// TIA Portal V20 export
// export: Created 2025-12-01T14:56:51.5395909Z, ExportSetting None, DisplayName Totally Integrated Automation Portal, DisplayVersion V20 Update 3, DisplayName TIA Portal Openness, DisplayVersion V20 Update 3, DisplayName TIA Portal Version Control Interface, DisplayVersion V20 Update 3, DisplayName STEP 7 Professional, DisplayVersion V20 Update 3, DisplayName STEP 7 Safety, DisplayVersion V20 Update 2, DisplayName WinCC Basic/Comfort/Advanced, DisplayVersion V20 Update 3, DisplayName WinCC Professional, DisplayVersion V20 Update 3, DisplayName WinCC Unified, DisplayVersion V20 Update 3
FUNCTION_BLOCK "FB351_DesRemontador_Remontador_Horquilla"   // FB351, LAD
TITLE = Control del Ramal de Salidas
{ S7_Optimized_Access := 'FALSE' }
AUTHOR : REFORMAR
NAME : 20160211
VERSION : 3.1
// Dani Palacios: Modificación octubre 2017 para poder desabilitar la maquina con un bit (por ejemplo en la puesta a punto si no esta montada o en el simulador)
// La modificación esta sin probar y es todo lo relativo a la variable Maquina_Desabilitada
// (bloqueo evolución desde etapa 0, bloqueo activación salidas en etapa 0 , fin vi sin mirar detectores y activación posición de reposo sin mirar detectores y variabkles de fin de movimiento).
// ES RESPONSABILIDAD DEL QUE DESABILITA LA MAQUINA QUE ESTA ESTE EN UNA POSICION QUE PERMITA EL MOVIMIENTO DE LAS CARGAS A TRAVES DE ELLA
// stored: AutoNumber false, SetENOAutomatically false
   VAR_INPUT
      Maquina : UInt;   // Numero de Maquina (Mesa)
      Error_Tx : Bool;   // Error en el Tx
      EnTension : Bool;   // Existe Tension en la Mesa
      MAQx_Desabilitada : Bool;   // Config MAQ. >>> DesHabilitada
      TipoPaleta : Bool;   // Si 1, EUR. Si 0, medio paleta
      Termico_Elevacion : Bool;   // Termico de la Elevacion
      Termico_Horquilla : Bool;   // Termico de la Horquilla
      ParElevacion_ErrorRotura : Bool;
      pHsMx : Bool;   // pHs de la Mesa
      EnMovimiento_Tx : Bool;   // En Movimiento Tx
      ELEV_SegUp : Bool;   // ELEV >> Seguridad Up
      ELEV_SegDw : Bool;   // ELEV >> Seguridad Down
      ELEV_PosUp : Bool;   // ELEV >> Posicion Up
      ELEV_PosMid : Bool;   // ELEV >> Posicion Midle
      ELEV_PosDw : Bool;   // ELEV >> Posicion Down
      ELEV_EnMovimiento : Bool;   // ELEV >> En Movimiento
      HORQ_SegRecogida : Bool;   // HORQ >> Seguridad Atras
      HORQ_SegExtendida : Bool;   // HORQ >> Seguridad Adelante
      HORQ_Recogida : Bool;   // HORQ >> Posicion Atras
      HORQ_Medio : Bool;   // HORQ >> Posicion Medio
      HORQ_Extendida : Bool;   // HORQ >> Posicion Adelante
      HORQ_CV_Recogida : Bool;   // HORQ >> Cambio de Velocidad Atras
      HORQ_CV_Medio : Bool;   // HORQ >> Cambio de Velocidad Medio
      HORQ_CV_Extendida : Bool;   // HORQ >> Cambio de Velocidad Adelante
      HORQ_EnMovimiento : Bool;   // HORQ >> En Movimiento
      Elev_Carga_OK : Bool;
      RH_PasarReposo : Bool;   // Interlock >> Pasar a Reposo
      RH_SubirPaleta : Bool;   // Interlock >> Subir Paleta
      RH_DejarPaleta : Bool;   // Interlock >> Dejar Paleta
      RH_RemontarPaleta : Bool;   // Interlock >> Remontar Paleta
      RH_DesRemontarPaleta : Bool;   // Interlock >> DesRemontar Paleta
      V_TIM_EstabilidadMov : Time;   // TIM de Estabilidad de los Mov.
      V_TOut_Elevacion : Int := 7000;   // TimeOut del Mov. de Elevacion
      V_TOut_Horquillado : Int := 7000;   // TimeOut del Mov. de Horquillado
   END_VAR
   VAR_OUTPUT
      RH_Quieto : Bool;   // Interlock >> Quieto
      RH_FinMovimiento : Bool;   // Interlock >> Fin del Movimiento
   END_VAR
   VAR
      Rh_ET00 : Bool;
      Rh_ET100 : Bool;
      Rh_ET101 : Bool;
      Rh_ET102 : Bool;
      Rh_ET103 : Bool;
      Rh_ET104 : Bool;
      Rh_ET105 : Bool;
      Rh_ET106 : Bool;
      Rh_ET107 : Bool;
      Rh_ET108 : Bool;
      Rh_ET109 : Bool;
      Rh_ET11 : Bool;
      Rh_ET12 : Bool;
      Rh_ET13 : Bool;
      Rh_ET14 : Bool;
      Rh_ET15 : Bool;
      Rh_ET16 : Bool;
      Rh_ET21 : Bool;
      Rh_ET22 : Bool;
      Rh_ET23 : Bool;
      Rh_ET24 : Bool;
      Rh_ET31 : Bool;
      Rh_ET32 : Bool;
      Rh_ET41 : Bool;
      Rh_ET42 : Bool;
      Rh_ET43 : Bool;
      Rh_ET44 : Bool;
      Rh_ET51 : Bool;
      Rh_ET52 : Bool;
      Rh_ET53 : Bool;
      PosicionConocida : Bool;
      STAT_Quieto : Bool;   // Interna >> Quieto la Maquina
      STAT_FinMovimiento : Bool;   // Interna >> Fin de Movimiento
      CambioDir_SubidaBajada : Bool;   // Interna >> Cambio de Dir. Subida o Bajada
      MA_Ir_Up : Bool;
      MA_Ir_Dw : Bool;
      MA_Ir_Mid_Bajando : Bool;
      MA_Ir_Mid_Subiendo : Bool;
      MA_Ir_Adelante : Bool;
      MA_Ir_Atras : Bool;
      HORQ_VelocidadRapida : Bool;
      TIM_EstabilidadMov { S7_SetPoint := 'True'} : TON_TIME;
      TMP_EnTension { S7_SetPoint := 'True'} : "FB910_CNT_UHS";
      TOut_Elevacion { S7_SetPoint := 'True'} : "FB910_CNT_UHS";
      TOut_Horquillado { S7_SetPoint := 'True'} : "FB910_CNT_UHS";
      Manual : "MoviManualMaquina_Remontador";
   END_VAR
   VAR_TEMP
      EstadoZona : "EstadoZona";   // Estado de Zona de la Mesa
      EstadoMAQ : "EstadoMaquina_Remontador";   // Estado del Vehiculo Inteliguente de la Maquina
      Aux_ET00 : Bool;
   END_VAR
BEGIN

REGION Network 1: INICIALIZAR - Recoger las Variables de Estado de la Maquina
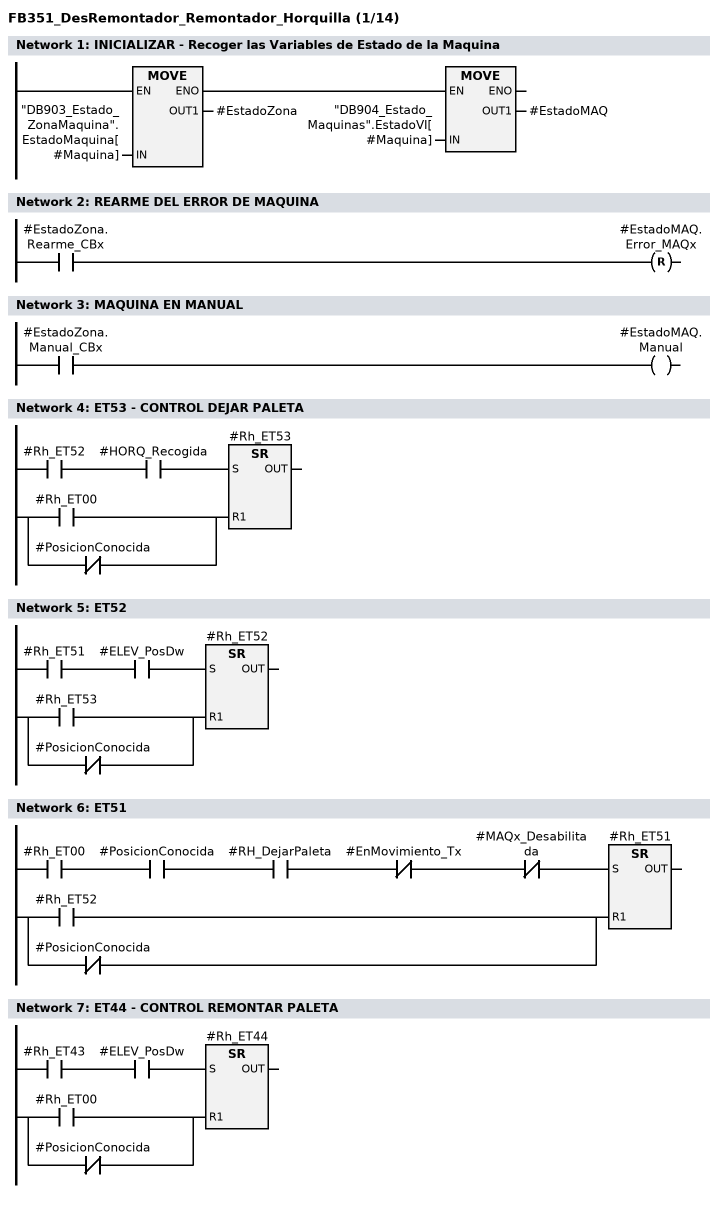
   RUNG wire#powerrail
      Move(in := "DB903_Estado_ZonaMaquina".EstadoMaquina[#Maquina], out1 => #EstadoZona)
      Move(in := "DB904_Estado_Maquinas".EstadoVI[#Maquina], out1 => #EstadoMAQ)
   END_RUNG
   // the same network as SCL:
   #EstadoZona := "DB903_Estado_ZonaMaquina".EstadoMaquina[#Maquina];
   #EstadoMAQ := "DB904_Estado_Maquinas".EstadoVI[#Maquina];
END_REGION

REGION Network 2: REARME DEL ERROR DE MAQUINA
   RUNG wire#powerrail
      Contact( #EstadoZona.Rearme_CBx )
      R_Coil( #EstadoMAQ.Error_MAQx )
   END_RUNG
   // the same network as SCL:
   IF #EstadoZona.Rearme_CBx THEN #EstadoMAQ.Error_MAQx := FALSE; END_IF;
END_REGION

REGION Network 3: MAQUINA EN MANUAL
   RUNG wire#powerrail
      Contact( #EstadoZona.Manual_CBx )
      Coil( #EstadoMAQ.Manual )
   END_RUNG
   // the same network as SCL:
   #EstadoMAQ.Manual := #EstadoZona.Manual_CBx;
END_REGION

REGION Network 4: ET53 - CONTROL DEJAR PALETA
   RUNG wire#powerrail
      Contact( #Rh_ET52 )
      Contact( #HORQ_Recogida )
      S_SR(operand := #Rh_ET53, r1 := wire#w1)
   END_RUNG
   RUNG wire#powerrail
      Contact( #Rh_ET00 )
   END_RUNG wire#w1
   RUNG wire#powerrail
      I_Contact( #PosicionConocida )
   END_RUNG wire#w1
   // the same network as SCL:
   IF #Rh_ET52 AND #HORQ_Recogida THEN
       #Rh_ET53 := TRUE;   // SR flip-flop
   END_IF;
   IF #Rh_ET00 OR NOT #PosicionConocida THEN #Rh_ET53 := FALSE; END_IF;
END_REGION

REGION Network 5: ET52
   RUNG wire#powerrail
      Contact( #Rh_ET51 )
      Contact( #ELEV_PosDw )
      S_SR(operand := #Rh_ET52, r1 := wire#w1)
   END_RUNG
   RUNG wire#powerrail
      Contact( #Rh_ET53 )
   END_RUNG wire#w1
   RUNG wire#powerrail
      I_Contact( #PosicionConocida )
   END_RUNG wire#w1
   // the same network as SCL:
   IF #Rh_ET51 AND #ELEV_PosDw THEN
       #Rh_ET52 := TRUE;   // SR flip-flop
   END_IF;
   IF #Rh_ET53 OR NOT #PosicionConocida THEN #Rh_ET52 := FALSE; END_IF;
END_REGION

REGION Network 6: ET51
   RUNG wire#powerrail
      Contact( #Rh_ET00 )
      Contact( #PosicionConocida )
      Contact( #RH_DejarPaleta )
      I_Contact( #EnMovimiento_Tx )
      I_Contact( #MAQx_Desabilitada )
      S_SR(operand := #Rh_ET51, r1 := wire#w1)
   END_RUNG
   RUNG wire#powerrail
      Contact( #Rh_ET52 )
   END_RUNG wire#w1
   RUNG wire#powerrail
      I_Contact( #PosicionConocida )
   END_RUNG wire#w1
   // the same network as SCL:
   IF #Rh_ET00 AND #PosicionConocida AND #RH_DejarPaleta AND NOT #EnMovimiento_Tx AND NOT #MAQx_Desabilitada THEN
       #Rh_ET51 := TRUE;   // SR flip-flop
   END_IF;
   IF #Rh_ET52 OR NOT #PosicionConocida THEN #Rh_ET51 := FALSE; END_IF;
END_REGION

REGION Network 7: ET44 - CONTROL REMONTAR PALETA
   RUNG wire#powerrail
      Contact( #Rh_ET43 )
      Contact( #ELEV_PosDw )
      S_SR(operand := #Rh_ET44, r1 := wire#w1)
   END_RUNG
   RUNG wire#powerrail
      Contact( #Rh_ET00 )
   END_RUNG wire#w1
   RUNG wire#powerrail
      I_Contact( #PosicionConocida )
   END_RUNG wire#w1
   // the same network as SCL:
   IF #Rh_ET43 AND #ELEV_PosDw THEN
       #Rh_ET44 := TRUE;   // SR flip-flop
   END_IF;
   IF #Rh_ET00 OR NOT #PosicionConocida THEN #Rh_ET44 := FALSE; END_IF;
END_REGION

REGION Network 8: ET43
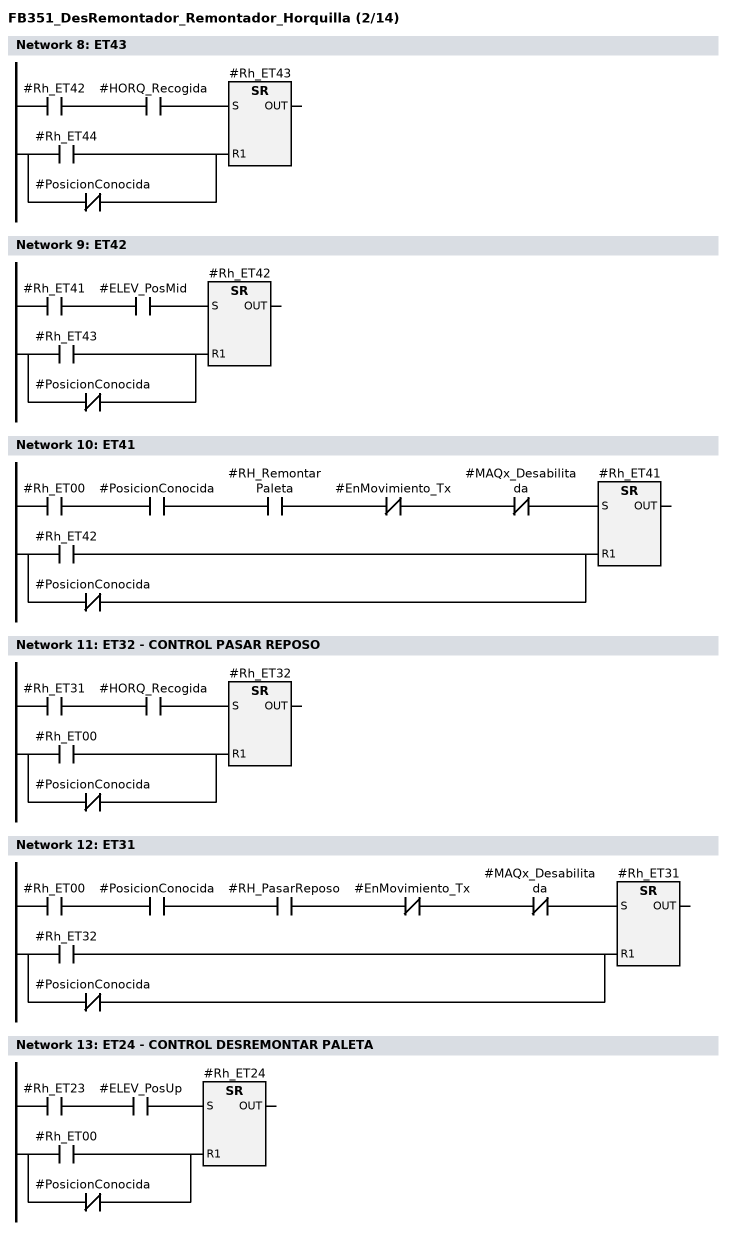
   RUNG wire#powerrail
      Contact( #Rh_ET42 )
      Contact( #HORQ_Recogida )
      S_SR(operand := #Rh_ET43, r1 := wire#w1)
   END_RUNG
   RUNG wire#powerrail
      Contact( #Rh_ET44 )
   END_RUNG wire#w1
   RUNG wire#powerrail
      I_Contact( #PosicionConocida )
   END_RUNG wire#w1
   // the same network as SCL:
   IF #Rh_ET42 AND #HORQ_Recogida THEN
       #Rh_ET43 := TRUE;   // SR flip-flop
   END_IF;
   IF #Rh_ET44 OR NOT #PosicionConocida THEN #Rh_ET43 := FALSE; END_IF;
END_REGION

REGION Network 9: ET42
   RUNG wire#powerrail
      Contact( #Rh_ET41 )
      Contact( #ELEV_PosMid )
      S_SR(operand := #Rh_ET42, r1 := wire#w1)
   END_RUNG
   RUNG wire#powerrail
      Contact( #Rh_ET43 )
   END_RUNG wire#w1
   RUNG wire#powerrail
      I_Contact( #PosicionConocida )
   END_RUNG wire#w1
   // the same network as SCL:
   IF #Rh_ET41 AND #ELEV_PosMid THEN
       #Rh_ET42 := TRUE;   // SR flip-flop
   END_IF;
   IF #Rh_ET43 OR NOT #PosicionConocida THEN #Rh_ET42 := FALSE; END_IF;
END_REGION

REGION Network 10: ET41
   RUNG wire#powerrail
      Contact( #Rh_ET00 )
      Contact( #PosicionConocida )
      Contact( #RH_RemontarPaleta )
      I_Contact( #EnMovimiento_Tx )
      I_Contact( #MAQx_Desabilitada )
      S_SR(operand := #Rh_ET41, r1 := wire#w1)
   END_RUNG
   RUNG wire#powerrail
      Contact( #Rh_ET42 )
   END_RUNG wire#w1
   RUNG wire#powerrail
      I_Contact( #PosicionConocida )
   END_RUNG wire#w1
   // the same network as SCL:
   IF #Rh_ET00 AND #PosicionConocida AND #RH_RemontarPaleta AND NOT #EnMovimiento_Tx AND NOT #MAQx_Desabilitada THEN
       #Rh_ET41 := TRUE;   // SR flip-flop
   END_IF;
   IF #Rh_ET42 OR NOT #PosicionConocida THEN #Rh_ET41 := FALSE; END_IF;
END_REGION

REGION Network 11: ET32 - CONTROL PASAR REPOSO
   RUNG wire#powerrail
      Contact( #Rh_ET31 )
      Contact( #HORQ_Recogida )
      S_SR(operand := #Rh_ET32, r1 := wire#w1)
   END_RUNG
   RUNG wire#powerrail
      Contact( #Rh_ET00 )
   END_RUNG wire#w1
   RUNG wire#powerrail
      I_Contact( #PosicionConocida )
   END_RUNG wire#w1
   // the same network as SCL:
   IF #Rh_ET31 AND #HORQ_Recogida THEN
       #Rh_ET32 := TRUE;   // SR flip-flop
   END_IF;
   IF #Rh_ET00 OR NOT #PosicionConocida THEN #Rh_ET32 := FALSE; END_IF;
END_REGION

REGION Network 12: ET31
   RUNG wire#powerrail
      Contact( #Rh_ET00 )
      Contact( #PosicionConocida )
      Contact( #RH_PasarReposo )
      I_Contact( #EnMovimiento_Tx )
      I_Contact( #MAQx_Desabilitada )
      S_SR(operand := #Rh_ET31, r1 := wire#w1)
   END_RUNG
   RUNG wire#powerrail
      Contact( #Rh_ET32 )
   END_RUNG wire#w1
   RUNG wire#powerrail
      I_Contact( #PosicionConocida )
   END_RUNG wire#w1
   // the same network as SCL:
   IF #Rh_ET00 AND #PosicionConocida AND #RH_PasarReposo AND NOT #EnMovimiento_Tx AND NOT #MAQx_Desabilitada THEN
       #Rh_ET31 := TRUE;   // SR flip-flop
   END_IF;
   IF #Rh_ET32 OR NOT #PosicionConocida THEN #Rh_ET31 := FALSE; END_IF;
END_REGION

REGION Network 13: ET24 - CONTROL DESREMONTAR PALETA
   RUNG wire#powerrail
      Contact( #Rh_ET23 )
      Contact( #ELEV_PosUp )
      S_SR(operand := #Rh_ET24, r1 := wire#w1)
   END_RUNG
   RUNG wire#powerrail
      Contact( #Rh_ET00 )
   END_RUNG wire#w1
   RUNG wire#powerrail
      I_Contact( #PosicionConocida )
   END_RUNG wire#w1
   // the same network as SCL:
   IF #Rh_ET23 AND #ELEV_PosUp THEN
       #Rh_ET24 := TRUE;   // SR flip-flop
   END_IF;
   IF #Rh_ET00 OR NOT #PosicionConocida THEN #Rh_ET24 := FALSE; END_IF;
END_REGION

REGION Network 14: ET23
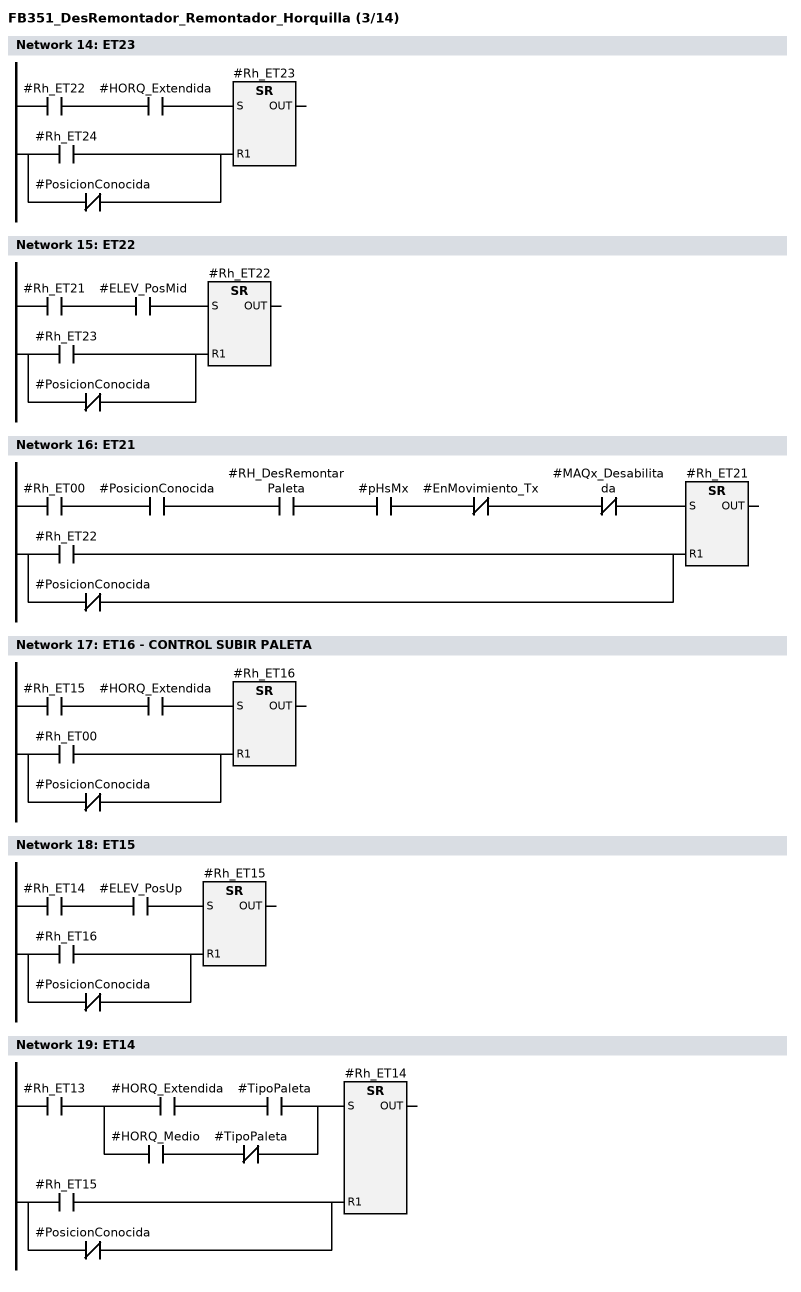
   RUNG wire#powerrail
      Contact( #Rh_ET22 )
      Contact( #HORQ_Extendida )
      S_SR(operand := #Rh_ET23, r1 := wire#w1)
   END_RUNG
   RUNG wire#powerrail
      Contact( #Rh_ET24 )
   END_RUNG wire#w1
   RUNG wire#powerrail
      I_Contact( #PosicionConocida )
   END_RUNG wire#w1
   // the same network as SCL:
   IF #Rh_ET22 AND #HORQ_Extendida THEN
       #Rh_ET23 := TRUE;   // SR flip-flop
   END_IF;
   IF #Rh_ET24 OR NOT #PosicionConocida THEN #Rh_ET23 := FALSE; END_IF;
END_REGION

REGION Network 15: ET22
   RUNG wire#powerrail
      Contact( #Rh_ET21 )
      Contact( #ELEV_PosMid )
      S_SR(operand := #Rh_ET22, r1 := wire#w1)
   END_RUNG
   RUNG wire#powerrail
      Contact( #Rh_ET23 )
   END_RUNG wire#w1
   RUNG wire#powerrail
      I_Contact( #PosicionConocida )
   END_RUNG wire#w1
   // the same network as SCL:
   IF #Rh_ET21 AND #ELEV_PosMid THEN
       #Rh_ET22 := TRUE;   // SR flip-flop
   END_IF;
   IF #Rh_ET23 OR NOT #PosicionConocida THEN #Rh_ET22 := FALSE; END_IF;
END_REGION

REGION Network 16: ET21
   RUNG wire#powerrail
      Contact( #Rh_ET00 )
      Contact( #PosicionConocida )
      Contact( #RH_DesRemontarPaleta )
      Contact( #pHsMx )
      I_Contact( #EnMovimiento_Tx )
      I_Contact( #MAQx_Desabilitada )
      S_SR(operand := #Rh_ET21, r1 := wire#w1)
   END_RUNG
   RUNG wire#powerrail
      Contact( #Rh_ET22 )
   END_RUNG wire#w1
   RUNG wire#powerrail
      I_Contact( #PosicionConocida )
   END_RUNG wire#w1
   // the same network as SCL:
   IF #Rh_ET00 AND #PosicionConocida AND #RH_DesRemontarPaleta AND #pHsMx AND NOT #EnMovimiento_Tx AND NOT #MAQx_Desabilitada THEN
       #Rh_ET21 := TRUE;   // SR flip-flop
   END_IF;
   IF #Rh_ET22 OR NOT #PosicionConocida THEN #Rh_ET21 := FALSE; END_IF;
END_REGION

REGION Network 17: ET16 - CONTROL SUBIR PALETA
   RUNG wire#powerrail
      Contact( #Rh_ET15 )
      Contact( #HORQ_Extendida )
      S_SR(operand := #Rh_ET16, r1 := wire#w1)
   END_RUNG
   RUNG wire#powerrail
      Contact( #Rh_ET00 )
   END_RUNG wire#w1
   RUNG wire#powerrail
      I_Contact( #PosicionConocida )
   END_RUNG wire#w1
   // the same network as SCL:
   IF #Rh_ET15 AND #HORQ_Extendida THEN
       #Rh_ET16 := TRUE;   // SR flip-flop
   END_IF;
   IF #Rh_ET00 OR NOT #PosicionConocida THEN #Rh_ET16 := FALSE; END_IF;
END_REGION

REGION Network 18: ET15
   RUNG wire#powerrail
      Contact( #Rh_ET14 )
      Contact( #ELEV_PosUp )
      S_SR(operand := #Rh_ET15, r1 := wire#w1)
   END_RUNG
   RUNG wire#powerrail
      Contact( #Rh_ET16 )
   END_RUNG wire#w1
   RUNG wire#powerrail
      I_Contact( #PosicionConocida )
   END_RUNG wire#w1
   // the same network as SCL:
   IF #Rh_ET14 AND #ELEV_PosUp THEN
       #Rh_ET15 := TRUE;   // SR flip-flop
   END_IF;
   IF #Rh_ET16 OR NOT #PosicionConocida THEN #Rh_ET15 := FALSE; END_IF;
END_REGION

REGION Network 19: ET14
   RUNG wire#powerrail
      Contact( #Rh_ET13 )
      wire#w1
      Contact( #HORQ_Extendida )
      Contact( #TipoPaleta )
      wire#w2
      S_SR(operand := #Rh_ET14, r1 := wire#w3)
   END_RUNG
   RUNG wire#w1
      Contact( #HORQ_Medio )
      I_Contact( #TipoPaleta )
   END_RUNG wire#w2
   RUNG wire#powerrail
      Contact( #Rh_ET15 )
   END_RUNG wire#w3
   RUNG wire#powerrail
      I_Contact( #PosicionConocida )
   END_RUNG wire#w3
   // the same network as SCL:
   IF #Rh_ET13 AND ((#HORQ_Extendida AND #TipoPaleta) OR (#HORQ_Medio AND NOT #TipoPaleta)) THEN
       #Rh_ET14 := TRUE;   // SR flip-flop
   END_IF;
   IF #Rh_ET15 OR NOT #PosicionConocida THEN #Rh_ET14 := FALSE; END_IF;
END_REGION

REGION Network 20: ET13
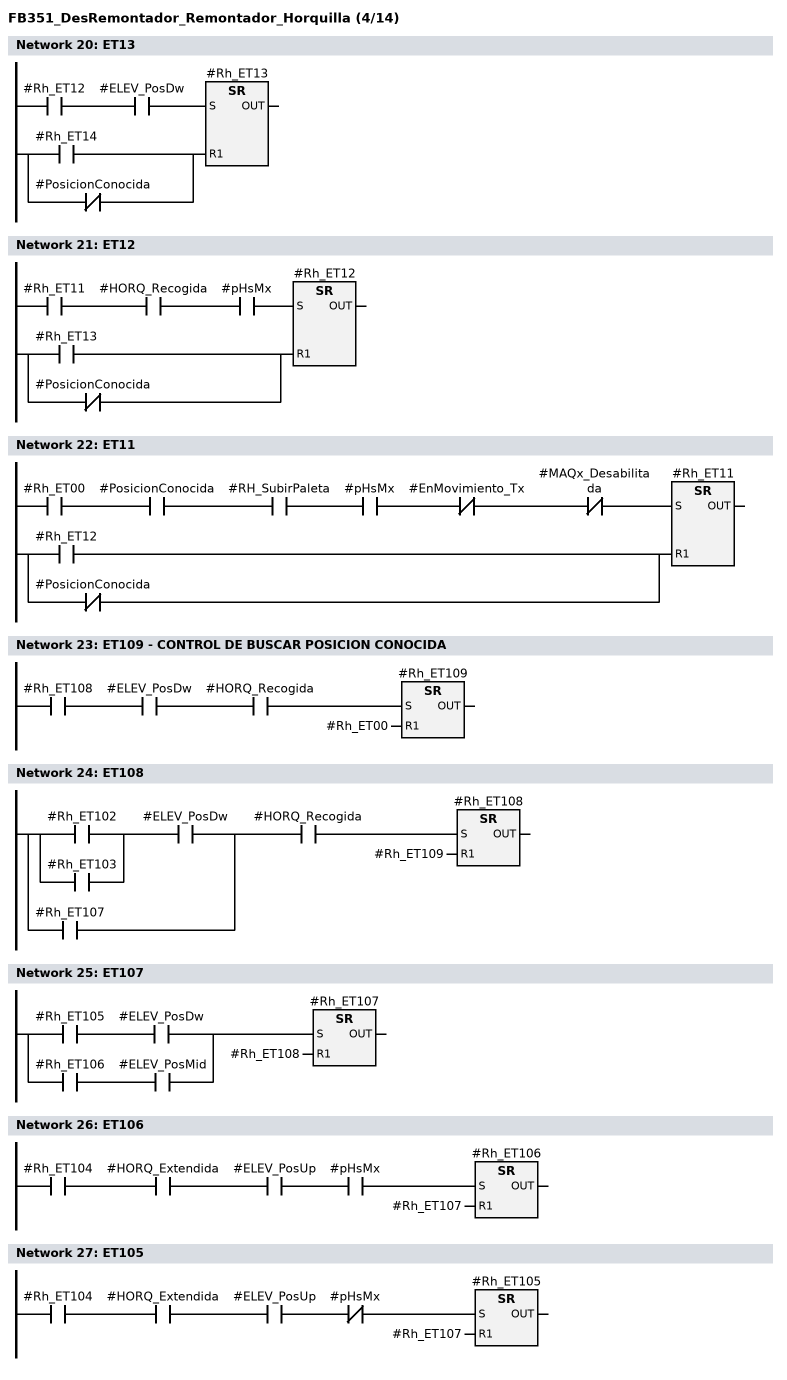
   RUNG wire#powerrail
      Contact( #Rh_ET12 )
      Contact( #ELEV_PosDw )
      S_SR(operand := #Rh_ET13, r1 := wire#w1)
   END_RUNG
   RUNG wire#powerrail
      Contact( #Rh_ET14 )
   END_RUNG wire#w1
   RUNG wire#powerrail
      I_Contact( #PosicionConocida )
   END_RUNG wire#w1
   // the same network as SCL:
   IF #Rh_ET12 AND #ELEV_PosDw THEN
       #Rh_ET13 := TRUE;   // SR flip-flop
   END_IF;
   IF #Rh_ET14 OR NOT #PosicionConocida THEN #Rh_ET13 := FALSE; END_IF;
END_REGION

REGION Network 21: ET12
   RUNG wire#powerrail
      Contact( #Rh_ET11 )
      Contact( #HORQ_Recogida )
      Contact( #pHsMx )
      S_SR(operand := #Rh_ET12, r1 := wire#w1)
   END_RUNG
   RUNG wire#powerrail
      Contact( #Rh_ET13 )
   END_RUNG wire#w1
   RUNG wire#powerrail
      I_Contact( #PosicionConocida )
   END_RUNG wire#w1
   // the same network as SCL:
   IF #Rh_ET11 AND #HORQ_Recogida AND #pHsMx THEN
       #Rh_ET12 := TRUE;   // SR flip-flop
   END_IF;
   IF #Rh_ET13 OR NOT #PosicionConocida THEN #Rh_ET12 := FALSE; END_IF;
END_REGION

REGION Network 22: ET11
   RUNG wire#powerrail
      Contact( #Rh_ET00 )
      Contact( #PosicionConocida )
      Contact( #RH_SubirPaleta )
      Contact( #pHsMx )
      I_Contact( #EnMovimiento_Tx )
      I_Contact( #MAQx_Desabilitada )
      S_SR(operand := #Rh_ET11, r1 := wire#w1)
   END_RUNG
   RUNG wire#powerrail
      Contact( #Rh_ET12 )
   END_RUNG wire#w1
   RUNG wire#powerrail
      I_Contact( #PosicionConocida )
   END_RUNG wire#w1
   // the same network as SCL:
   IF #Rh_ET00 AND #PosicionConocida AND #RH_SubirPaleta AND #pHsMx AND NOT #EnMovimiento_Tx AND NOT #MAQx_Desabilitada THEN
       #Rh_ET11 := TRUE;   // SR flip-flop
   END_IF;
   IF #Rh_ET12 OR NOT #PosicionConocida THEN #Rh_ET11 := FALSE; END_IF;
END_REGION

REGION Network 23: ET109 - CONTROL DE BUSCAR POSICION CONOCIDA
   RUNG wire#powerrail
      Contact( #Rh_ET108 )
      Contact( #ELEV_PosDw )
      Contact( #HORQ_Recogida )
      S_SR(operand := #Rh_ET109, r1 := #Rh_ET00)
   END_RUNG
   // the same network as SCL:
   IF #Rh_ET108 AND #ELEV_PosDw AND #HORQ_Recogida THEN
       #Rh_ET109 := TRUE;   // SR flip-flop
   END_IF;
   IF #Rh_ET00 THEN #Rh_ET109 := FALSE; END_IF;
END_REGION

REGION Network 24: ET108
   RUNG wire#powerrail
      Contact( #Rh_ET102 )
      wire#w1
      Contact( #ELEV_PosDw )
      wire#w2
      Contact( #HORQ_Recogida )
      S_SR(operand := #Rh_ET108, r1 := #Rh_ET109)
   END_RUNG
   RUNG wire#powerrail
      Contact( #Rh_ET103 )
   END_RUNG wire#w1
   RUNG wire#powerrail
      Contact( #Rh_ET107 )
   END_RUNG wire#w2
   // the same network as SCL:
   IF (((#Rh_ET102 OR #Rh_ET103) AND #ELEV_PosDw) OR #Rh_ET107) AND #HORQ_Recogida THEN
       #Rh_ET108 := TRUE;   // SR flip-flop
   END_IF;
   IF #Rh_ET109 THEN #Rh_ET108 := FALSE; END_IF;
END_REGION

REGION Network 25: ET107
   RUNG wire#powerrail
      Contact( #Rh_ET105 )
      Contact( #ELEV_PosDw )
      wire#w1
      S_SR(operand := #Rh_ET107, r1 := #Rh_ET108)
   END_RUNG
   RUNG wire#powerrail
      Contact( #Rh_ET106 )
      Contact( #ELEV_PosMid )
   END_RUNG wire#w1
   // the same network as SCL:
   IF (#Rh_ET105 AND #ELEV_PosDw) OR (#Rh_ET106 AND #ELEV_PosMid) THEN
       #Rh_ET107 := TRUE;   // SR flip-flop
   END_IF;
   IF #Rh_ET108 THEN #Rh_ET107 := FALSE; END_IF;
END_REGION

REGION Network 26: ET106
   RUNG wire#powerrail
      Contact( #Rh_ET104 )
      Contact( #HORQ_Extendida )
      Contact( #ELEV_PosUp )
      Contact( #pHsMx )
      S_SR(operand := #Rh_ET106, r1 := #Rh_ET107)
   END_RUNG
   // the same network as SCL:
   IF #Rh_ET104 AND #HORQ_Extendida AND #ELEV_PosUp AND #pHsMx THEN
       #Rh_ET106 := TRUE;   // SR flip-flop
   END_IF;
   IF #Rh_ET107 THEN #Rh_ET106 := FALSE; END_IF;
END_REGION

REGION Network 27: ET105
   RUNG wire#powerrail
      Contact( #Rh_ET104 )
      Contact( #HORQ_Extendida )
      Contact( #ELEV_PosUp )
      I_Contact( #pHsMx )
      S_SR(operand := #Rh_ET105, r1 := #Rh_ET107)
   END_RUNG
   // the same network as SCL:
   IF #Rh_ET104 AND #HORQ_Extendida AND #ELEV_PosUp AND NOT #pHsMx THEN
       #Rh_ET105 := TRUE;   // SR flip-flop
   END_IF;
   IF #Rh_ET107 THEN #Rh_ET105 := FALSE; END_IF;
END_REGION

REGION Network 28: ET104
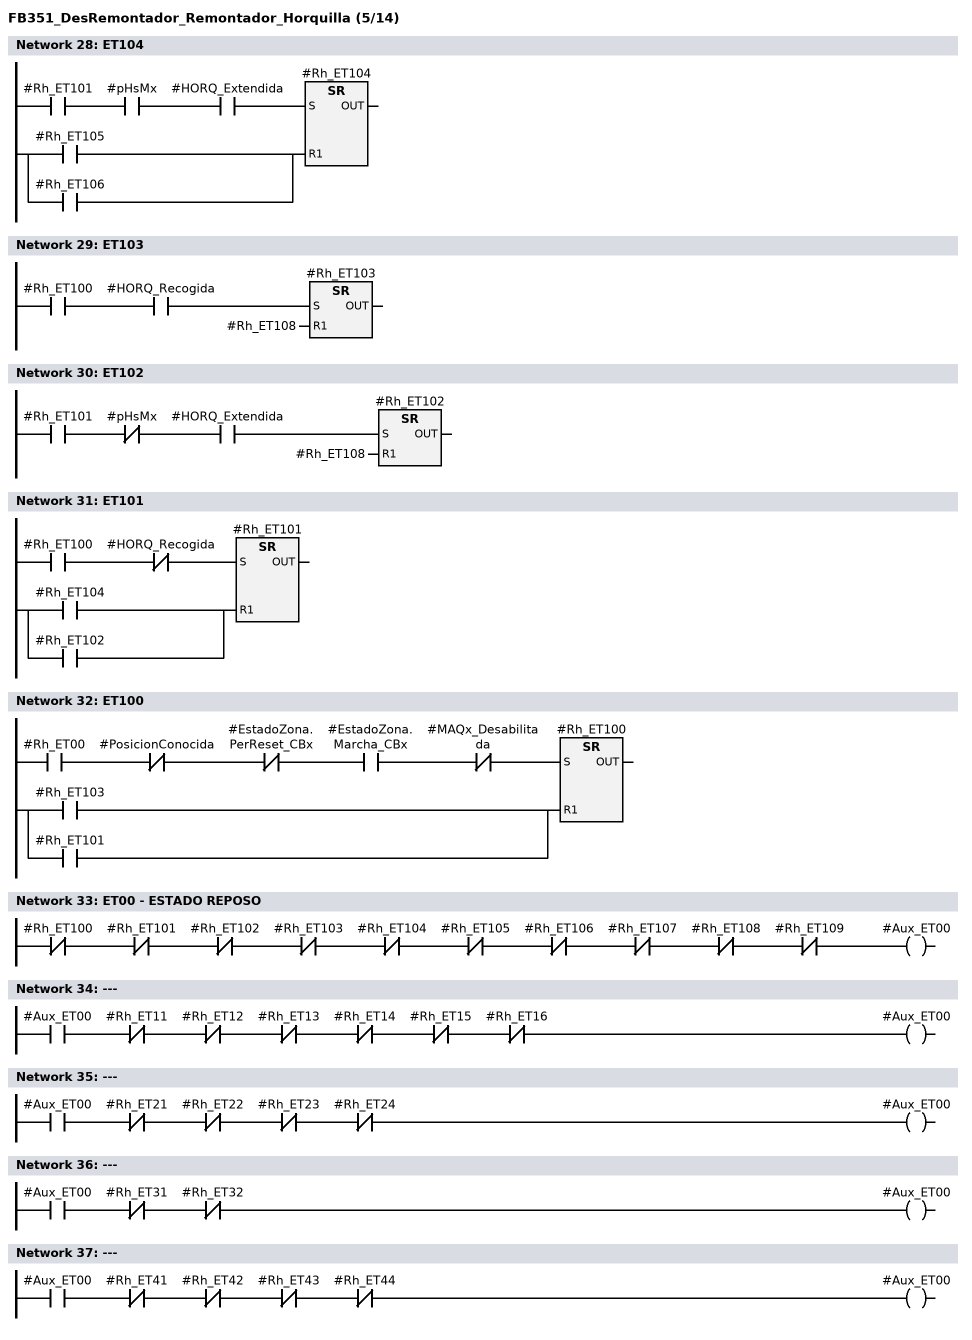
   RUNG wire#powerrail
      Contact( #Rh_ET101 )
      Contact( #pHsMx )
      Contact( #HORQ_Extendida )
      S_SR(operand := #Rh_ET104, r1 := wire#w1)
   END_RUNG
   RUNG wire#powerrail
      Contact( #Rh_ET105 )
   END_RUNG wire#w1
   RUNG wire#powerrail
      Contact( #Rh_ET106 )
   END_RUNG wire#w1
   // the same network as SCL:
   IF #Rh_ET101 AND #pHsMx AND #HORQ_Extendida THEN
       #Rh_ET104 := TRUE;   // SR flip-flop
   END_IF;
   IF #Rh_ET105 OR #Rh_ET106 THEN #Rh_ET104 := FALSE; END_IF;
END_REGION

REGION Network 29: ET103
   RUNG wire#powerrail
      Contact( #Rh_ET100 )
      Contact( #HORQ_Recogida )
      S_SR(operand := #Rh_ET103, r1 := #Rh_ET108)
   END_RUNG
   // the same network as SCL:
   IF #Rh_ET100 AND #HORQ_Recogida THEN
       #Rh_ET103 := TRUE;   // SR flip-flop
   END_IF;
   IF #Rh_ET108 THEN #Rh_ET103 := FALSE; END_IF;
END_REGION

REGION Network 30: ET102
   RUNG wire#powerrail
      Contact( #Rh_ET101 )
      I_Contact( #pHsMx )
      Contact( #HORQ_Extendida )
      S_SR(operand := #Rh_ET102, r1 := #Rh_ET108)
   END_RUNG
   // the same network as SCL:
   IF #Rh_ET101 AND NOT #pHsMx AND #HORQ_Extendida THEN
       #Rh_ET102 := TRUE;   // SR flip-flop
   END_IF;
   IF #Rh_ET108 THEN #Rh_ET102 := FALSE; END_IF;
END_REGION

REGION Network 31: ET101
   RUNG wire#powerrail
      Contact( #Rh_ET100 )
      I_Contact( #HORQ_Recogida )
      S_SR(operand := #Rh_ET101, r1 := wire#w1)
   END_RUNG
   RUNG wire#powerrail
      Contact( #Rh_ET104 )
   END_RUNG wire#w1
   RUNG wire#powerrail
      Contact( #Rh_ET102 )
   END_RUNG wire#w1
   // the same network as SCL:
   IF #Rh_ET100 AND NOT #HORQ_Recogida THEN
       #Rh_ET101 := TRUE;   // SR flip-flop
   END_IF;
   IF #Rh_ET104 OR #Rh_ET102 THEN #Rh_ET101 := FALSE; END_IF;
END_REGION

REGION Network 32: ET100
   RUNG wire#powerrail
      Contact( #Rh_ET00 )
      I_Contact( #PosicionConocida )
      I_Contact( #EstadoZona.PerReset_CBx )
      Contact( #EstadoZona.Marcha_CBx )
      I_Contact( #MAQx_Desabilitada )
      S_SR(operand := #Rh_ET100, r1 := wire#w1)
   END_RUNG
   RUNG wire#powerrail
      Contact( #Rh_ET103 )
   END_RUNG wire#w1
   RUNG wire#powerrail
      Contact( #Rh_ET101 )
   END_RUNG wire#w1
   // the same network as SCL:
   IF #Rh_ET00 AND NOT #PosicionConocida AND NOT #EstadoZona.PerReset_CBx AND #EstadoZona.Marcha_CBx AND NOT #MAQx_Desabilitada THEN
       #Rh_ET100 := TRUE;   // SR flip-flop
   END_IF;
   IF #Rh_ET103 OR #Rh_ET101 THEN #Rh_ET100 := FALSE; END_IF;
END_REGION

REGION Network 33: ET00 - ESTADO REPOSO
   RUNG wire#powerrail
      I_Contact( #Rh_ET100 )
      I_Contact( #Rh_ET101 )
      I_Contact( #Rh_ET102 )
      I_Contact( #Rh_ET103 )
      I_Contact( #Rh_ET104 )
      I_Contact( #Rh_ET105 )
      I_Contact( #Rh_ET106 )
      I_Contact( #Rh_ET107 )
      I_Contact( #Rh_ET108 )
      I_Contact( #Rh_ET109 )
      Coil( #Aux_ET00 )
   END_RUNG
   // the same network as SCL:
   #Aux_ET00 := NOT #Rh_ET100 AND NOT #Rh_ET101 AND NOT #Rh_ET102 AND NOT #Rh_ET103 AND NOT #Rh_ET104 AND NOT #Rh_ET105 AND NOT #Rh_ET106 AND NOT #Rh_ET107 AND NOT #Rh_ET108 AND NOT #Rh_ET109;
END_REGION

REGION Network 34: ---
   RUNG wire#powerrail
      Contact( #Aux_ET00 )
      I_Contact( #Rh_ET11 )
      I_Contact( #Rh_ET12 )
      I_Contact( #Rh_ET13 )
      I_Contact( #Rh_ET14 )
      I_Contact( #Rh_ET15 )
      I_Contact( #Rh_ET16 )
      Coil( #Aux_ET00 )
   END_RUNG
   // the same network as SCL:
   #Aux_ET00 := #Aux_ET00 AND NOT #Rh_ET11 AND NOT #Rh_ET12 AND NOT #Rh_ET13 AND NOT #Rh_ET14 AND NOT #Rh_ET15 AND NOT #Rh_ET16;
END_REGION

REGION Network 35: ---
   RUNG wire#powerrail
      Contact( #Aux_ET00 )
      I_Contact( #Rh_ET21 )
      I_Contact( #Rh_ET22 )
      I_Contact( #Rh_ET23 )
      I_Contact( #Rh_ET24 )
      Coil( #Aux_ET00 )
   END_RUNG
   // the same network as SCL:
   #Aux_ET00 := #Aux_ET00 AND NOT #Rh_ET21 AND NOT #Rh_ET22 AND NOT #Rh_ET23 AND NOT #Rh_ET24;
END_REGION

REGION Network 36: ---
   RUNG wire#powerrail
      Contact( #Aux_ET00 )
      I_Contact( #Rh_ET31 )
      I_Contact( #Rh_ET32 )
      Coil( #Aux_ET00 )
   END_RUNG
   // the same network as SCL:
   #Aux_ET00 := #Aux_ET00 AND NOT #Rh_ET31 AND NOT #Rh_ET32;
END_REGION

REGION Network 37: ---
   RUNG wire#powerrail
      Contact( #Aux_ET00 )
      I_Contact( #Rh_ET41 )
      I_Contact( #Rh_ET42 )
      I_Contact( #Rh_ET43 )
      I_Contact( #Rh_ET44 )
      Coil( #Aux_ET00 )
   END_RUNG
   // the same network as SCL:
   #Aux_ET00 := #Aux_ET00 AND NOT #Rh_ET41 AND NOT #Rh_ET42 AND NOT #Rh_ET43 AND NOT #Rh_ET44;
END_REGION

REGION Network 38: ---
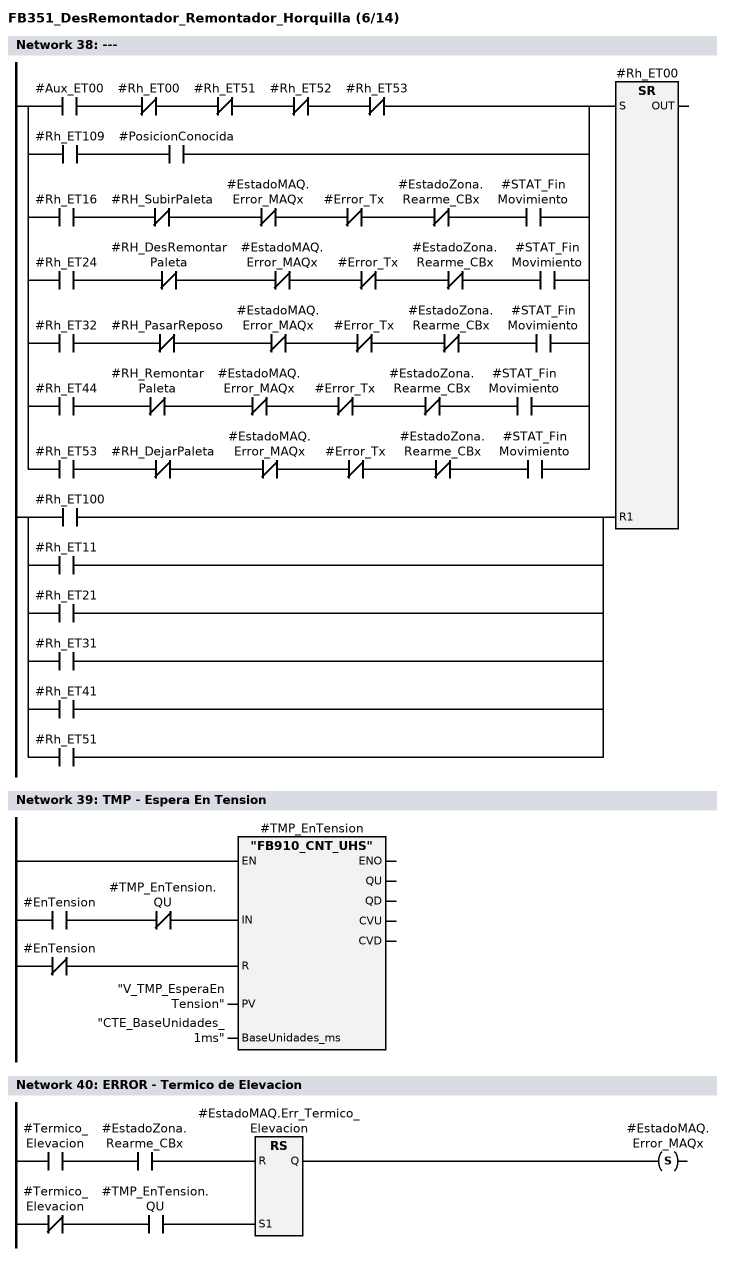
   RUNG wire#powerrail
      Contact( #Aux_ET00 )
      I_Contact( #Rh_ET00 )
      I_Contact( #Rh_ET51 )
      I_Contact( #Rh_ET52 )
      I_Contact( #Rh_ET53 )
      wire#w1
      S_SR(operand := #Rh_ET00, r1 := wire#w2)
   END_RUNG
   RUNG wire#powerrail
      Contact( #Rh_ET109 )
      Contact( #PosicionConocida )
   END_RUNG wire#w1
   RUNG wire#powerrail
      Contact( #Rh_ET16 )
      I_Contact( #RH_SubirPaleta )
      I_Contact( #EstadoMAQ.Error_MAQx )
      I_Contact( #Error_Tx )
      I_Contact( #EstadoZona.Rearme_CBx )
      Contact( #STAT_FinMovimiento )
   END_RUNG wire#w1
   RUNG wire#powerrail
      Contact( #Rh_ET24 )
      I_Contact( #RH_DesRemontarPaleta )
      I_Contact( #EstadoMAQ.Error_MAQx )
      I_Contact( #Error_Tx )
      I_Contact( #EstadoZona.Rearme_CBx )
      Contact( #STAT_FinMovimiento )
   END_RUNG wire#w1
   RUNG wire#powerrail
      Contact( #Rh_ET32 )
      I_Contact( #RH_PasarReposo )
      I_Contact( #EstadoMAQ.Error_MAQx )
      I_Contact( #Error_Tx )
      I_Contact( #EstadoZona.Rearme_CBx )
      Contact( #STAT_FinMovimiento )
   END_RUNG wire#w1
   RUNG wire#powerrail
      Contact( #Rh_ET44 )
      I_Contact( #RH_RemontarPaleta )
      I_Contact( #EstadoMAQ.Error_MAQx )
      I_Contact( #Error_Tx )
      I_Contact( #EstadoZona.Rearme_CBx )
      Contact( #STAT_FinMovimiento )
   END_RUNG wire#w1
   RUNG wire#powerrail
      Contact( #Rh_ET53 )
      I_Contact( #RH_DejarPaleta )
      I_Contact( #EstadoMAQ.Error_MAQx )
      I_Contact( #Error_Tx )
      I_Contact( #EstadoZona.Rearme_CBx )
      Contact( #STAT_FinMovimiento )
   END_RUNG wire#w1
   RUNG wire#powerrail
      Contact( #Rh_ET100 )
   END_RUNG wire#w2
   RUNG wire#powerrail
      Contact( #Rh_ET11 )
   END_RUNG wire#w2
   RUNG wire#powerrail
      Contact( #Rh_ET21 )
   END_RUNG wire#w2
   RUNG wire#powerrail
      Contact( #Rh_ET31 )
   END_RUNG wire#w2
   RUNG wire#powerrail
      Contact( #Rh_ET41 )
   END_RUNG wire#w2
   RUNG wire#powerrail
      Contact( #Rh_ET51 )
   END_RUNG wire#w2
   // the same network as SCL:
   IF (#Aux_ET00 AND NOT #Rh_ET00 AND NOT #Rh_ET51 AND NOT #Rh_ET52 AND NOT #Rh_ET53) OR (#Rh_ET109 AND #PosicionConocida) OR (#Rh_ET16 AND NOT #RH_SubirPaleta AND NOT #EstadoMAQ.Error_MAQx AND NOT #Error_Tx AND NOT #EstadoZona.Rearme_CBx AND #STAT_FinMovimiento) OR (#Rh_ET24 AND NOT #RH_DesRemontarPaleta AND NOT #EstadoMAQ.Error_MAQx AND NOT #Error_Tx AND NOT #EstadoZona.Rearme_CBx AND #STAT_FinMovimiento) OR (#Rh_ET32 AND NOT #RH_PasarReposo AND NOT #EstadoMAQ.Error_MAQx AND NOT #Error_Tx AND NOT #EstadoZona.Rearme_CBx AND #STAT_FinMovimiento) OR (#Rh_ET44 AND NOT #RH_RemontarPaleta AND NOT #EstadoMAQ.Error_MAQx AND NOT #Error_Tx AND NOT #EstadoZona.Rearme_CBx AND #STAT_FinMovimiento) OR (#Rh_ET53 AND NOT #RH_DejarPaleta AND NOT #EstadoMAQ.Error_MAQx AND NOT #Error_Tx AND NOT #EstadoZona.Rearme_CBx AND #STAT_FinMovimiento) THEN
       #Rh_ET00 := TRUE;   // SR flip-flop
   END_IF;
   IF #Rh_ET100 OR #Rh_ET11 OR #Rh_ET21 OR #Rh_ET31 OR #Rh_ET41 OR #Rh_ET51 THEN #Rh_ET00 := FALSE; END_IF;
END_REGION

REGION Network 39: TMP - Espera En Tension
   RUNG wire#powerrail
      #TMP_EnTension(IN := wire#w1, R := wire#w2, PV := "V_TMP_EsperaEnTension", BaseUnidades_ms := "CTE_BaseUnidades_1ms", QU =>, QD =>, CVU =>, CVD =>)
   END_RUNG
   RUNG wire#powerrail
      Contact( #EnTension )
      I_Contact( #TMP_EnTension.QU )
   END_RUNG wire#w1
   RUNG wire#powerrail
      I_Contact( #EnTension )
   END_RUNG wire#w2
   // the same network as SCL:
   #TMP_EnTension(IN := #EnTension AND NOT #TMP_EnTension.QU,   // "FB910_CNT_UHS"
                  R := NOT #EnTension,
                  PV := "V_TMP_EsperaEnTension",
                  BaseUnidades_ms := "CTE_BaseUnidades_1ms");
END_REGION

REGION Network 40: ERROR - Termico de Elevacion
   RUNG wire#powerrail
      Contact( #Termico_Elevacion )
      Contact( #EstadoZona.Rearme_CBx )
      S_RS(operand := #EstadoMAQ.Err_Termico_Elevacion, s1 := wire#w1)
      S_Coil( #EstadoMAQ.Error_MAQx )
   END_RUNG
   RUNG wire#powerrail
      I_Contact( #Termico_Elevacion )
      Contact( #TMP_EnTension.QU )
   END_RUNG wire#w1
   // the same network as SCL:
   IF #Termico_Elevacion AND #EstadoZona.Rearme_CBx THEN
       #EstadoMAQ.Err_Termico_Elevacion := FALSE;   // RS flip-flop
   END_IF;
   IF NOT #Termico_Elevacion AND #TMP_EnTension.QU THEN #EstadoMAQ.Err_Termico_Elevacion := TRUE; END_IF;
   IF #EstadoMAQ.Err_Termico_Elevacion THEN #EstadoMAQ.Error_MAQx := TRUE; END_IF;
END_REGION

REGION Network 41: ERROR - Termico de Horquilla
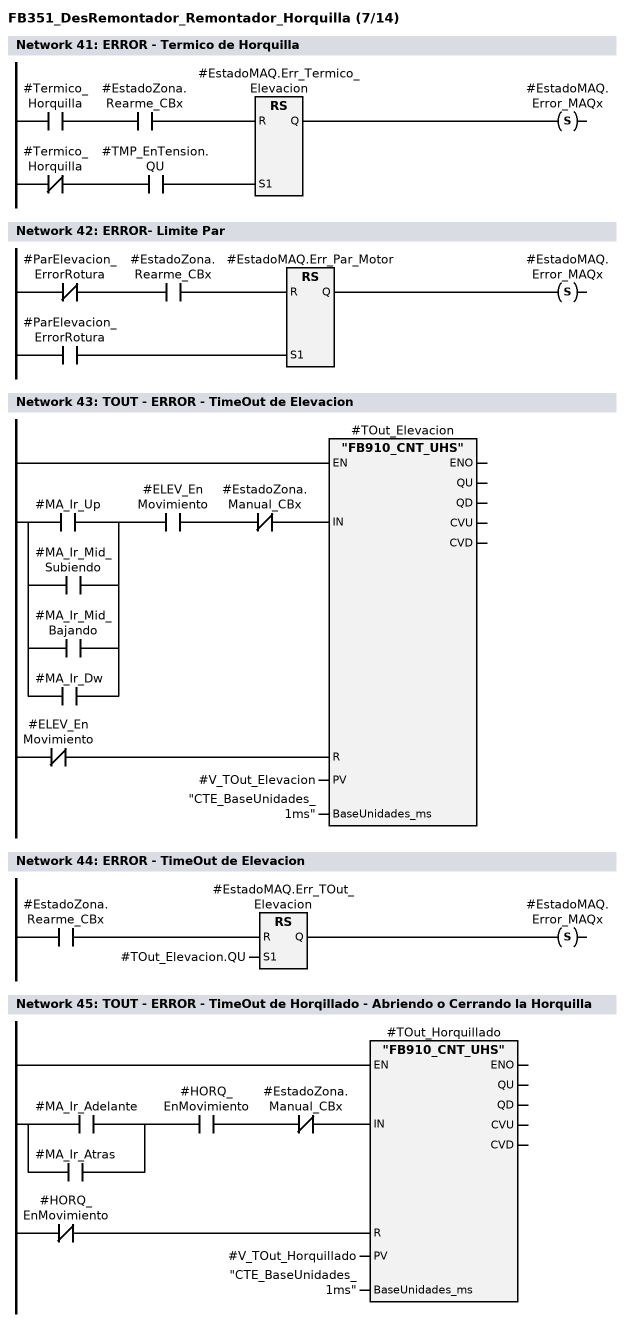
   RUNG wire#powerrail
      Contact( #Termico_Horquilla )
      Contact( #EstadoZona.Rearme_CBx )
      S_RS(operand := #EstadoMAQ.Err_Termico_Elevacion, s1 := wire#w1)
      S_Coil( #EstadoMAQ.Error_MAQx )
   END_RUNG
   RUNG wire#powerrail
      I_Contact( #Termico_Horquilla )
      Contact( #TMP_EnTension.QU )
   END_RUNG wire#w1
   // the same network as SCL:
   IF #Termico_Horquilla AND #EstadoZona.Rearme_CBx THEN
       #EstadoMAQ.Err_Termico_Elevacion := FALSE;   // RS flip-flop
   END_IF;
   IF NOT #Termico_Horquilla AND #TMP_EnTension.QU THEN #EstadoMAQ.Err_Termico_Elevacion := TRUE; END_IF;
   IF #EstadoMAQ.Err_Termico_Elevacion THEN #EstadoMAQ.Error_MAQx := TRUE; END_IF;
END_REGION

REGION Network 42: ERROR- Limite Par
   RUNG wire#powerrail
      I_Contact( #ParElevacion_ErrorRotura )
      Contact( #EstadoZona.Rearme_CBx )
      S_RS(operand := #EstadoMAQ.Err_Par_Motor, s1 := wire#w1)
      S_Coil( #EstadoMAQ.Error_MAQx )
   END_RUNG
   RUNG wire#powerrail
      Contact( #ParElevacion_ErrorRotura )
   END_RUNG wire#w1
   // the same network as SCL:
   IF NOT #ParElevacion_ErrorRotura AND #EstadoZona.Rearme_CBx THEN
       #EstadoMAQ.Err_Par_Motor := FALSE;   // RS flip-flop
   END_IF;
   IF #ParElevacion_ErrorRotura THEN #EstadoMAQ.Err_Par_Motor := TRUE; END_IF;
   IF #EstadoMAQ.Err_Par_Motor THEN #EstadoMAQ.Error_MAQx := TRUE; END_IF;
END_REGION

REGION Network 43: TOUT - ERROR - TimeOut de Elevacion
   RUNG wire#powerrail
      #TOut_Elevacion(IN := wire#w2, R := wire#w3, PV := #V_TOut_Elevacion, BaseUnidades_ms := "CTE_BaseUnidades_1ms", QU =>, QD =>, CVU =>, CVD =>)
   END_RUNG
   RUNG wire#powerrail
      Contact( #MA_Ir_Up )
      wire#w1
      Contact( #ELEV_EnMovimiento )
      I_Contact( #EstadoZona.Manual_CBx )
   END_RUNG wire#w2
   RUNG wire#powerrail
      Contact( #MA_Ir_Mid_Subiendo )
   END_RUNG wire#w1
   RUNG wire#powerrail
      Contact( #MA_Ir_Mid_Bajando )
   END_RUNG wire#w1
   RUNG wire#powerrail
      Contact( #MA_Ir_Dw )
   END_RUNG wire#w1
   RUNG wire#powerrail
      I_Contact( #ELEV_EnMovimiento )
   END_RUNG wire#w3
   // the same network as SCL:
   #TOut_Elevacion(IN := (#MA_Ir_Up OR #MA_Ir_Mid_Subiendo OR #MA_Ir_Mid_Bajando OR #MA_Ir_Dw) AND #ELEV_EnMovimiento AND NOT #EstadoZona.Manual_CBx,   // "FB910_CNT_UHS"
                   R := NOT #ELEV_EnMovimiento,
                   PV := #V_TOut_Elevacion,
                   BaseUnidades_ms := "CTE_BaseUnidades_1ms");
END_REGION

REGION Network 44: ERROR - TimeOut de Elevacion
   RUNG wire#powerrail
      Contact( #EstadoZona.Rearme_CBx )
      S_RS(operand := #EstadoMAQ.Err_TOut_Elevacion, s1 := #TOut_Elevacion.QU)
      S_Coil( #EstadoMAQ.Error_MAQx )
   END_RUNG
   // the same network as SCL:
   IF #EstadoZona.Rearme_CBx THEN
       #EstadoMAQ.Err_TOut_Elevacion := FALSE;   // RS flip-flop
   END_IF;
   IF #TOut_Elevacion.QU THEN #EstadoMAQ.Err_TOut_Elevacion := TRUE; END_IF;
   IF #EstadoMAQ.Err_TOut_Elevacion THEN #EstadoMAQ.Error_MAQx := TRUE; END_IF;
END_REGION

REGION Network 45: TOUT - ERROR - TimeOut de Horqillado - Abriendo o Cerrando la Horquilla
   RUNG wire#powerrail
      #TOut_Horquillado(IN := wire#w2, R := wire#w3, PV := #V_TOut_Horquillado, BaseUnidades_ms := "CTE_BaseUnidades_1ms", QU =>, QD =>, CVU =>, CVD =>)
   END_RUNG
   RUNG wire#powerrail
      Contact( #MA_Ir_Adelante )
      wire#w1
      Contact( #HORQ_EnMovimiento )
      I_Contact( #EstadoZona.Manual_CBx )
   END_RUNG wire#w2
   RUNG wire#powerrail
      Contact( #MA_Ir_Atras )
   END_RUNG wire#w1
   RUNG wire#powerrail
      I_Contact( #HORQ_EnMovimiento )
   END_RUNG wire#w3
   // the same network as SCL:
   #TOut_Horquillado(IN := (#MA_Ir_Adelante OR #MA_Ir_Atras) AND #HORQ_EnMovimiento AND NOT #EstadoZona.Manual_CBx,   // "FB910_CNT_UHS"
                     R := NOT #HORQ_EnMovimiento,
                     PV := #V_TOut_Horquillado,
                     BaseUnidades_ms := "CTE_BaseUnidades_1ms");
END_REGION

REGION Network 46: ERROR - TimeOut de Horqillado - Abriendo la Horquilla
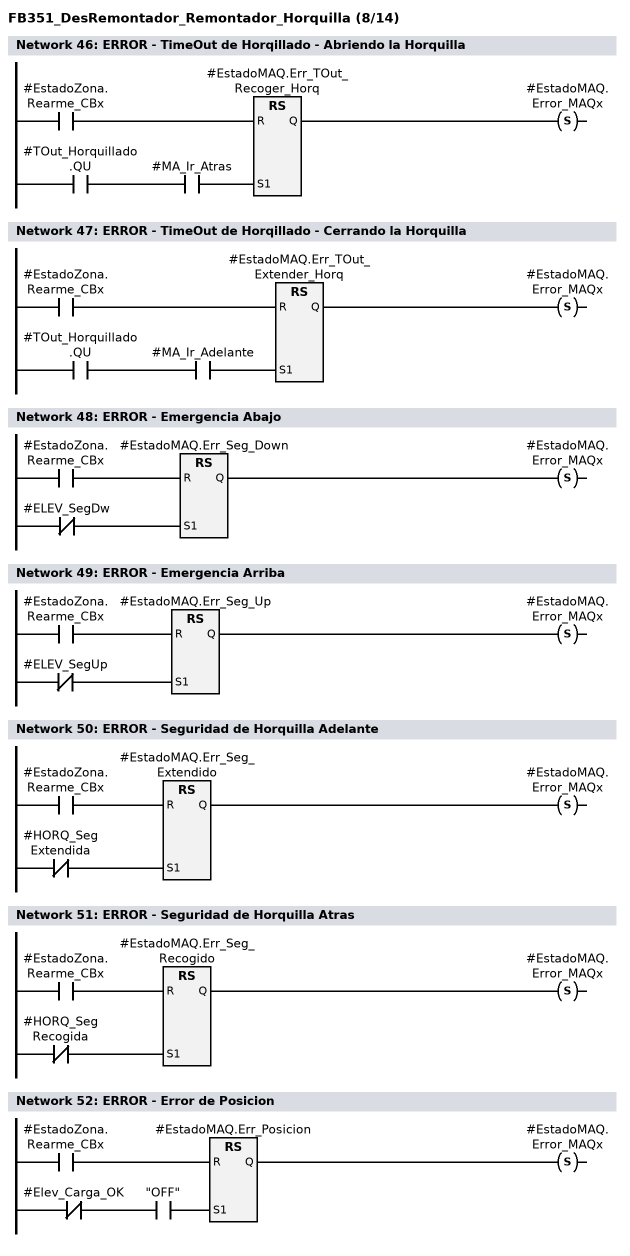
   RUNG wire#powerrail
      Contact( #EstadoZona.Rearme_CBx )
      S_RS(operand := #EstadoMAQ.Err_TOut_Recoger_Horq, s1 := wire#w1)
      S_Coil( #EstadoMAQ.Error_MAQx )
   END_RUNG
   RUNG wire#powerrail
      Contact( #TOut_Horquillado.QU )
      Contact( #MA_Ir_Atras )
   END_RUNG wire#w1
   // the same network as SCL:
   IF #EstadoZona.Rearme_CBx THEN
       #EstadoMAQ.Err_TOut_Recoger_Horq := FALSE;   // RS flip-flop
   END_IF;
   IF #TOut_Horquillado.QU AND #MA_Ir_Atras THEN #EstadoMAQ.Err_TOut_Recoger_Horq := TRUE; END_IF;
   IF #EstadoMAQ.Err_TOut_Recoger_Horq THEN #EstadoMAQ.Error_MAQx := TRUE; END_IF;
END_REGION

REGION Network 47: ERROR - TimeOut de Horqillado - Cerrando la Horquilla
   RUNG wire#powerrail
      Contact( #EstadoZona.Rearme_CBx )
      S_RS(operand := #EstadoMAQ.Err_TOut_Extender_Horq, s1 := wire#w1)
      S_Coil( #EstadoMAQ.Error_MAQx )
   END_RUNG
   RUNG wire#powerrail
      Contact( #TOut_Horquillado.QU )
      Contact( #MA_Ir_Adelante )
   END_RUNG wire#w1
   // the same network as SCL:
   IF #EstadoZona.Rearme_CBx THEN
       #EstadoMAQ.Err_TOut_Extender_Horq := FALSE;   // RS flip-flop
   END_IF;
   IF #TOut_Horquillado.QU AND #MA_Ir_Adelante THEN #EstadoMAQ.Err_TOut_Extender_Horq := TRUE; END_IF;
   IF #EstadoMAQ.Err_TOut_Extender_Horq THEN #EstadoMAQ.Error_MAQx := TRUE; END_IF;
END_REGION

REGION Network 48: ERROR - Emergencia Abajo
   RUNG wire#powerrail
      Contact( #EstadoZona.Rearme_CBx )
      S_RS(operand := #EstadoMAQ.Err_Seg_Down, s1 := wire#w1)
      S_Coil( #EstadoMAQ.Error_MAQx )
   END_RUNG
   RUNG wire#powerrail
      I_Contact( #ELEV_SegDw )
   END_RUNG wire#w1
   // the same network as SCL:
   IF #EstadoZona.Rearme_CBx THEN
       #EstadoMAQ.Err_Seg_Down := FALSE;   // RS flip-flop
   END_IF;
   IF NOT #ELEV_SegDw THEN #EstadoMAQ.Err_Seg_Down := TRUE; END_IF;
   IF #EstadoMAQ.Err_Seg_Down THEN #EstadoMAQ.Error_MAQx := TRUE; END_IF;
END_REGION

REGION Network 49: ERROR - Emergencia Arriba
   RUNG wire#powerrail
      Contact( #EstadoZona.Rearme_CBx )
      S_RS(operand := #EstadoMAQ.Err_Seg_Up, s1 := wire#w1)
      S_Coil( #EstadoMAQ.Error_MAQx )
   END_RUNG
   RUNG wire#powerrail
      I_Contact( #ELEV_SegUp )
   END_RUNG wire#w1
   // the same network as SCL:
   IF #EstadoZona.Rearme_CBx THEN
       #EstadoMAQ.Err_Seg_Up := FALSE;   // RS flip-flop
   END_IF;
   IF NOT #ELEV_SegUp THEN #EstadoMAQ.Err_Seg_Up := TRUE; END_IF;
   IF #EstadoMAQ.Err_Seg_Up THEN #EstadoMAQ.Error_MAQx := TRUE; END_IF;
END_REGION

REGION Network 50: ERROR - Seguridad de Horquilla Adelante
   RUNG wire#powerrail
      Contact( #EstadoZona.Rearme_CBx )
      S_RS(operand := #EstadoMAQ.Err_Seg_Extendido, s1 := wire#w1)
      S_Coil( #EstadoMAQ.Error_MAQx )
   END_RUNG
   RUNG wire#powerrail
      I_Contact( #HORQ_SegExtendida )
   END_RUNG wire#w1
   // the same network as SCL:
   IF #EstadoZona.Rearme_CBx THEN
       #EstadoMAQ.Err_Seg_Extendido := FALSE;   // RS flip-flop
   END_IF;
   IF NOT #HORQ_SegExtendida THEN #EstadoMAQ.Err_Seg_Extendido := TRUE; END_IF;
   IF #EstadoMAQ.Err_Seg_Extendido THEN #EstadoMAQ.Error_MAQx := TRUE; END_IF;
END_REGION

REGION Network 51: ERROR - Seguridad de Horquilla Atras
   RUNG wire#powerrail
      Contact( #EstadoZona.Rearme_CBx )
      S_RS(operand := #EstadoMAQ.Err_Seg_Recogido, s1 := wire#w1)
      S_Coil( #EstadoMAQ.Error_MAQx )
   END_RUNG
   RUNG wire#powerrail
      I_Contact( #HORQ_SegRecogida )
   END_RUNG wire#w1
   // the same network as SCL:
   IF #EstadoZona.Rearme_CBx THEN
       #EstadoMAQ.Err_Seg_Recogido := FALSE;   // RS flip-flop
   END_IF;
   IF NOT #HORQ_SegRecogida THEN #EstadoMAQ.Err_Seg_Recogido := TRUE; END_IF;
   IF #EstadoMAQ.Err_Seg_Recogido THEN #EstadoMAQ.Error_MAQx := TRUE; END_IF;
END_REGION

REGION Network 52: ERROR - Error de Posicion
   RUNG wire#powerrail
      Contact( #EstadoZona.Rearme_CBx )
      S_RS(operand := #EstadoMAQ.Err_Posicion, s1 := wire#w1)
      S_Coil( #EstadoMAQ.Error_MAQx )
   END_RUNG
   RUNG wire#powerrail
      I_Contact( #Elev_Carga_OK )
      Contact( "OFF" )
   END_RUNG wire#w1
   // the same network as SCL:
   IF #EstadoZona.Rearme_CBx THEN
       #EstadoMAQ.Err_Posicion := FALSE;   // RS flip-flop
   END_IF;
   IF NOT #Elev_Carga_OK AND "OFF" THEN #EstadoMAQ.Err_Posicion := TRUE; END_IF;
   IF #EstadoMAQ.Err_Posicion THEN #EstadoMAQ.Error_MAQx := TRUE; END_IF;
END_REGION

REGION Network 53: Error Carga
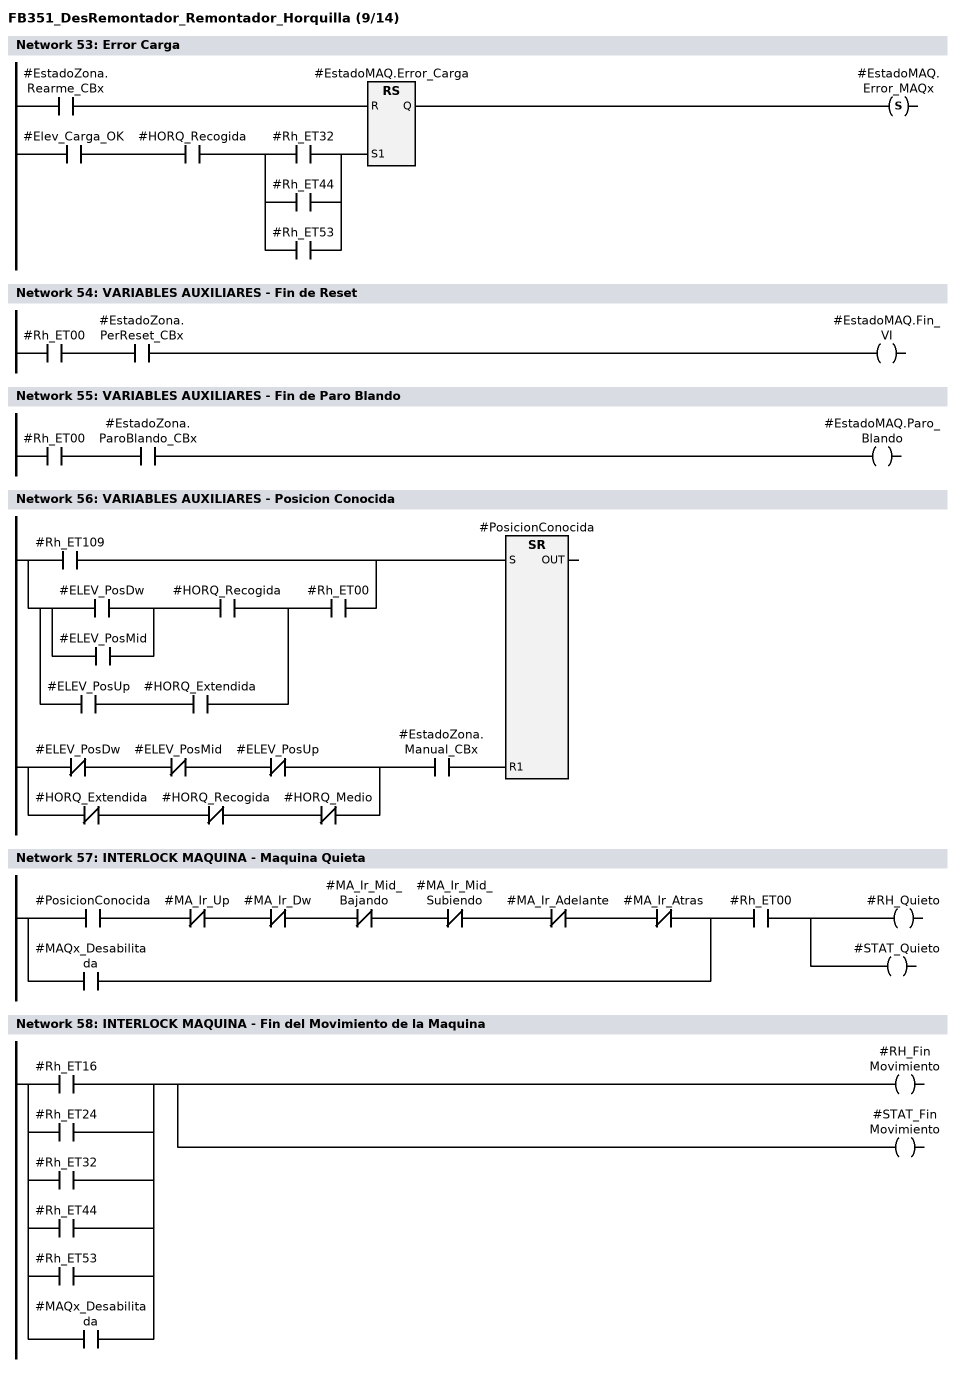
   RUNG wire#powerrail
      Contact( #EstadoZona.Rearme_CBx )
      S_RS(operand := #EstadoMAQ.Error_Carga, s1 := wire#w2)
      S_Coil( #EstadoMAQ.Error_MAQx )
   END_RUNG
   RUNG wire#powerrail
      Contact( #Elev_Carga_OK )
      Contact( #HORQ_Recogida )
      wire#w1
      Contact( #Rh_ET32 )
   END_RUNG wire#w2
   RUNG wire#w1
      Contact( #Rh_ET44 )
   END_RUNG wire#w2
   RUNG wire#w1
      Contact( #Rh_ET53 )
   END_RUNG wire#w2
   // the same network as SCL:
   IF #EstadoZona.Rearme_CBx THEN
       #EstadoMAQ.Error_Carga := FALSE;   // RS flip-flop
   END_IF;
   IF #Elev_Carga_OK AND #HORQ_Recogida AND (#Rh_ET32 OR #Rh_ET44 OR #Rh_ET53) THEN
       #EstadoMAQ.Error_Carga := TRUE;
   END_IF;
   IF #EstadoMAQ.Error_Carga THEN #EstadoMAQ.Error_MAQx := TRUE; END_IF;
END_REGION

REGION Network 54: VARIABLES AUXILIARES - Fin de Reset
   RUNG wire#powerrail
      Contact( #Rh_ET00 )
      Contact( #EstadoZona.PerReset_CBx )
      Coil( #EstadoMAQ.Fin_VI )
   END_RUNG
   // the same network as SCL:
   #EstadoMAQ.Fin_VI := #Rh_ET00 AND #EstadoZona.PerReset_CBx;
END_REGION

REGION Network 55: VARIABLES AUXILIARES - Fin de Paro Blando
   RUNG wire#powerrail
      Contact( #Rh_ET00 )
      Contact( #EstadoZona.ParoBlando_CBx )
      Coil( #EstadoMAQ.Paro_Blando )
   END_RUNG
   // the same network as SCL:
   #EstadoMAQ.Paro_Blando := #Rh_ET00 AND #EstadoZona.ParoBlando_CBx;
END_REGION

REGION Network 56: VARIABLES AUXILIARES - Posicion Conocida
   RUNG wire#powerrail
      Contact( #Rh_ET109 )
      wire#w1
      S_SR(operand := #PosicionConocida, r1 := wire#w5)
   END_RUNG
   RUNG wire#powerrail
      Contact( #ELEV_PosDw )
      wire#w2
      Contact( #HORQ_Recogida )
      wire#w3
      Contact( #Rh_ET00 )
   END_RUNG wire#w1
   RUNG wire#powerrail
      Contact( #ELEV_PosMid )
   END_RUNG wire#w2
   RUNG wire#powerrail
      Contact( #ELEV_PosUp )
      Contact( #HORQ_Extendida )
   END_RUNG wire#w3
   RUNG wire#powerrail
      I_Contact( #ELEV_PosDw )
      I_Contact( #ELEV_PosMid )
      I_Contact( #ELEV_PosUp )
      wire#w4
      Contact( #EstadoZona.Manual_CBx )
   END_RUNG wire#w5
   RUNG wire#powerrail
      I_Contact( #HORQ_Extendida )
      I_Contact( #HORQ_Recogida )
      I_Contact( #HORQ_Medio )
   END_RUNG wire#w4
   // the same network as SCL:
   IF #Rh_ET109 OR ((((#ELEV_PosDw OR #ELEV_PosMid) AND #HORQ_Recogida) OR (#ELEV_PosUp AND #HORQ_Extendida)) AND #Rh_ET00) THEN
       #PosicionConocida := TRUE;   // SR flip-flop
   END_IF;
   IF ((NOT #ELEV_PosDw AND NOT #ELEV_PosMid AND NOT #ELEV_PosUp) OR (NOT #HORQ_Extendida AND NOT #HORQ_Recogida AND NOT #HORQ_Medio)) AND #EstadoZona.Manual_CBx THEN
       #PosicionConocida := FALSE;
   END_IF;
END_REGION

REGION Network 57: INTERLOCK MAQUINA - Maquina Quieta
   RUNG wire#powerrail
      Contact( #PosicionConocida )
      I_Contact( #MA_Ir_Up )
      I_Contact( #MA_Ir_Dw )
      I_Contact( #MA_Ir_Mid_Bajando )
      I_Contact( #MA_Ir_Mid_Subiendo )
      I_Contact( #MA_Ir_Adelante )
      I_Contact( #MA_Ir_Atras )
      wire#w1
      Contact( #Rh_ET00 )
      wire#w2
      Coil( #RH_Quieto )
   END_RUNG
   RUNG wire#powerrail
      Contact( #MAQx_Desabilitada )
   END_RUNG wire#w1
   RUNG wire#w2
      Coil( #STAT_Quieto )
   END_RUNG
   // the same network as SCL:
   #RH_Quieto := ((#PosicionConocida AND NOT #MA_Ir_Up AND NOT #MA_Ir_Dw AND NOT #MA_Ir_Mid_Bajando AND NOT #MA_Ir_Mid_Subiendo AND NOT #MA_Ir_Adelante AND NOT #MA_Ir_Atras) OR #MAQx_Desabilitada) AND #Rh_ET00;
   #STAT_Quieto := #RH_Quieto;
END_REGION

REGION Network 58: INTERLOCK MAQUINA - Fin del Movimiento de la Maquina
   RUNG wire#powerrail
      Contact( #Rh_ET16 )
      wire#w1
      Coil( #RH_FinMovimiento )
   END_RUNG
   RUNG wire#powerrail
      Contact( #Rh_ET24 )
   END_RUNG wire#w1
   RUNG wire#powerrail
      Contact( #Rh_ET32 )
   END_RUNG wire#w1
   RUNG wire#powerrail
      Contact( #Rh_ET44 )
   END_RUNG wire#w1
   RUNG wire#powerrail
      Contact( #Rh_ET53 )
   END_RUNG wire#w1
   RUNG wire#powerrail
      Contact( #MAQx_Desabilitada )
   END_RUNG wire#w1
   RUNG wire#w1
      Coil( #STAT_FinMovimiento )
   END_RUNG
   // the same network as SCL:
   #RH_FinMovimiento := #Rh_ET16 OR #Rh_ET24 OR #Rh_ET32 OR #Rh_ET44 OR #Rh_ET53 OR #MAQx_Desabilitada;
   #STAT_FinMovimiento := #RH_FinMovimiento;
END_REGION

REGION Network 59: VARIABLES AUXILIARES - Cambiar de Direccion Buscando la Posicion Media
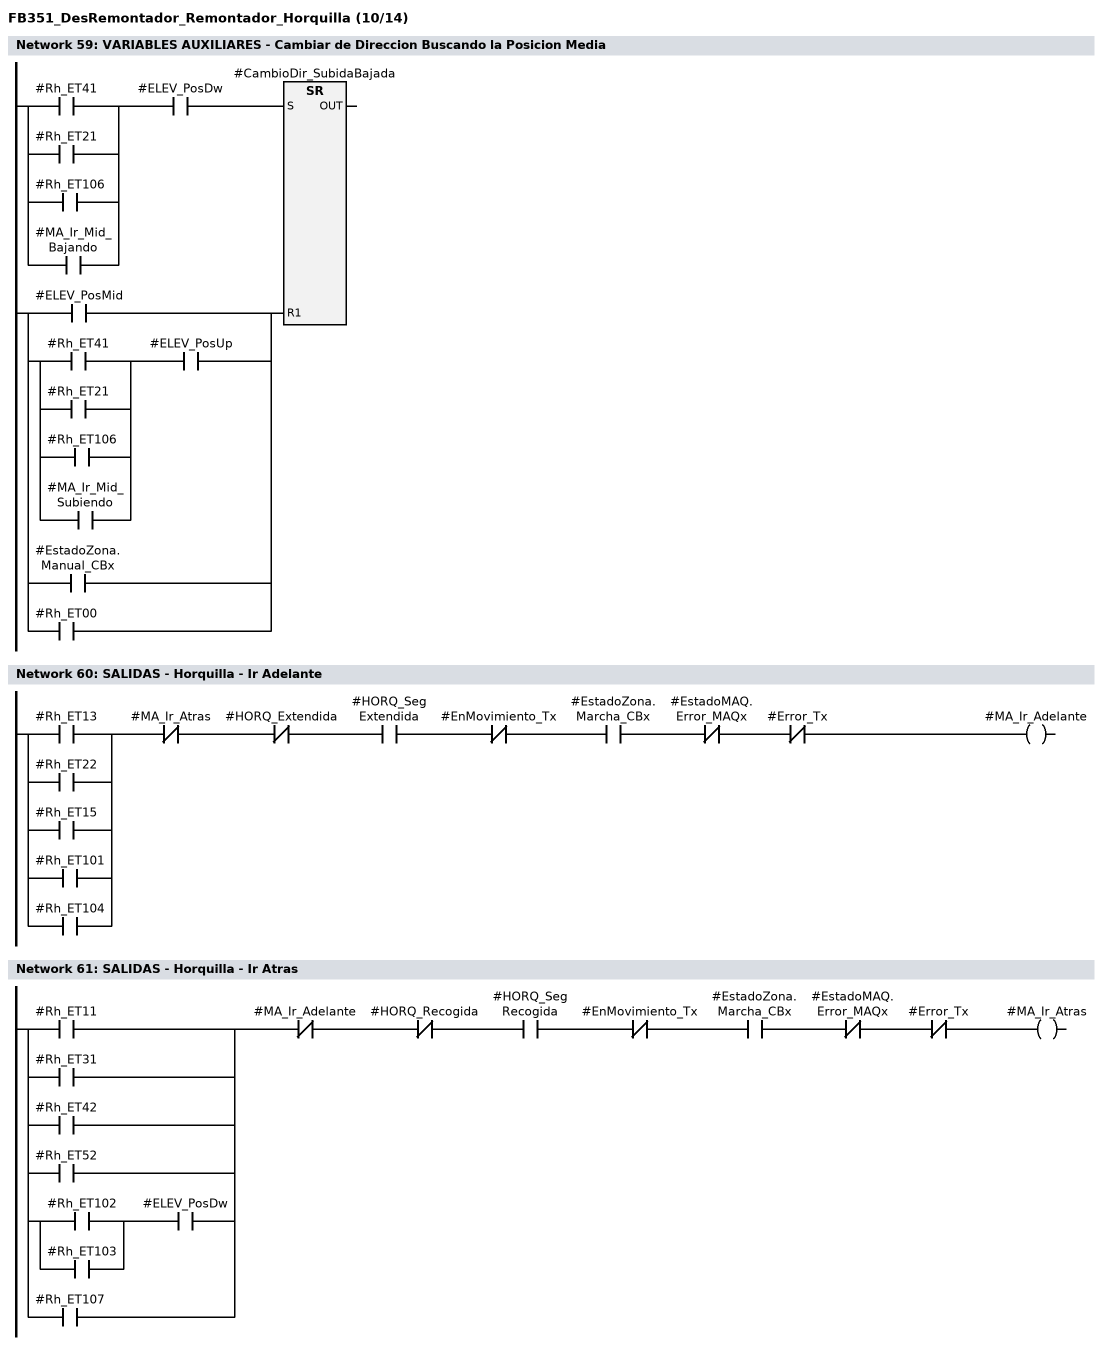
   RUNG wire#powerrail
      Contact( #Rh_ET41 )
      wire#w1
      Contact( #ELEV_PosDw )
      S_SR(operand := #CambioDir_SubidaBajada, r1 := wire#w3)
   END_RUNG
   RUNG wire#powerrail
      Contact( #Rh_ET21 )
   END_RUNG wire#w1
   RUNG wire#powerrail
      Contact( #Rh_ET106 )
   END_RUNG wire#w1
   RUNG wire#powerrail
      Contact( #MA_Ir_Mid_Bajando )
   END_RUNG wire#w1
   RUNG wire#powerrail
      Contact( #ELEV_PosMid )
   END_RUNG wire#w3
   RUNG wire#powerrail
      Contact( #Rh_ET41 )
      wire#w2
      Contact( #ELEV_PosUp )
   END_RUNG wire#w3
   RUNG wire#powerrail
      Contact( #Rh_ET21 )
   END_RUNG wire#w2
   RUNG wire#powerrail
      Contact( #Rh_ET106 )
   END_RUNG wire#w2
   RUNG wire#powerrail
      Contact( #MA_Ir_Mid_Subiendo )
   END_RUNG wire#w2
   RUNG wire#powerrail
      Contact( #EstadoZona.Manual_CBx )
   END_RUNG wire#w3
   RUNG wire#powerrail
      Contact( #Rh_ET00 )
   END_RUNG wire#w3
   // the same network as SCL:
   IF (#Rh_ET41 OR #Rh_ET21 OR #Rh_ET106 OR #MA_Ir_Mid_Bajando) AND #ELEV_PosDw THEN
       #CambioDir_SubidaBajada := TRUE;   // SR flip-flop
   END_IF;
   IF #ELEV_PosMid OR ((#Rh_ET41 OR #Rh_ET21 OR #Rh_ET106 OR #MA_Ir_Mid_Subiendo) AND #ELEV_PosUp) OR #EstadoZona.Manual_CBx OR #Rh_ET00 THEN
       #CambioDir_SubidaBajada := FALSE;
   END_IF;
END_REGION

REGION Network 60: SALIDAS - Horquilla - Ir Adelante
   RUNG wire#powerrail
      Contact( #Rh_ET13 )
      wire#w1
      I_Contact( #MA_Ir_Atras )
      I_Contact( #HORQ_Extendida )
      Contact( #HORQ_SegExtendida )
      I_Contact( #EnMovimiento_Tx )
      Contact( #EstadoZona.Marcha_CBx )
      I_Contact( #EstadoMAQ.Error_MAQx )
      I_Contact( #Error_Tx )
      Coil( #MA_Ir_Adelante )
   END_RUNG
   RUNG wire#powerrail
      Contact( #Rh_ET22 )
   END_RUNG wire#w1
   RUNG wire#powerrail
      Contact( #Rh_ET15 )
   END_RUNG wire#w1
   RUNG wire#powerrail
      Contact( #Rh_ET101 )
   END_RUNG wire#w1
   RUNG wire#powerrail
      Contact( #Rh_ET104 )
   END_RUNG wire#w1
   // the same network as SCL:
   #MA_Ir_Adelante := (#Rh_ET13 OR #Rh_ET22 OR #Rh_ET15 OR #Rh_ET101 OR #Rh_ET104) AND NOT #MA_Ir_Atras AND NOT #HORQ_Extendida AND #HORQ_SegExtendida AND NOT #EnMovimiento_Tx AND #EstadoZona.Marcha_CBx AND NOT #EstadoMAQ.Error_MAQx AND NOT #Error_Tx;
END_REGION

REGION Network 61: SALIDAS - Horquilla - Ir Atras
   RUNG wire#powerrail
      Contact( #Rh_ET11 )
      wire#w1
      I_Contact( #MA_Ir_Adelante )
      I_Contact( #HORQ_Recogida )
      Contact( #HORQ_SegRecogida )
      I_Contact( #EnMovimiento_Tx )
      Contact( #EstadoZona.Marcha_CBx )
      I_Contact( #EstadoMAQ.Error_MAQx )
      I_Contact( #Error_Tx )
      Coil( #MA_Ir_Atras )
   END_RUNG
   RUNG wire#powerrail
      Contact( #Rh_ET31 )
   END_RUNG wire#w1
   RUNG wire#powerrail
      Contact( #Rh_ET42 )
   END_RUNG wire#w1
   RUNG wire#powerrail
      Contact( #Rh_ET52 )
   END_RUNG wire#w1
   RUNG wire#powerrail
      Contact( #Rh_ET102 )
      wire#w2
      Contact( #ELEV_PosDw )
   END_RUNG wire#w1
   RUNG wire#powerrail
      Contact( #Rh_ET103 )
   END_RUNG wire#w2
   RUNG wire#powerrail
      Contact( #Rh_ET107 )
   END_RUNG wire#w1
   // the same network as SCL:
   #MA_Ir_Atras := (#Rh_ET11 OR #Rh_ET31 OR #Rh_ET42 OR #Rh_ET52 OR ((#Rh_ET102 OR #Rh_ET103) AND #ELEV_PosDw) OR #Rh_ET107) AND NOT #MA_Ir_Adelante AND NOT #HORQ_Recogida AND #HORQ_SegRecogida AND NOT #EnMovimiento_Tx AND #EstadoZona.Marcha_CBx AND NOT #EstadoMAQ.Error_MAQx AND NOT #Error_Tx;
END_REGION

REGION Network 62: SALIDAS - Elevacion - Ir DOWN
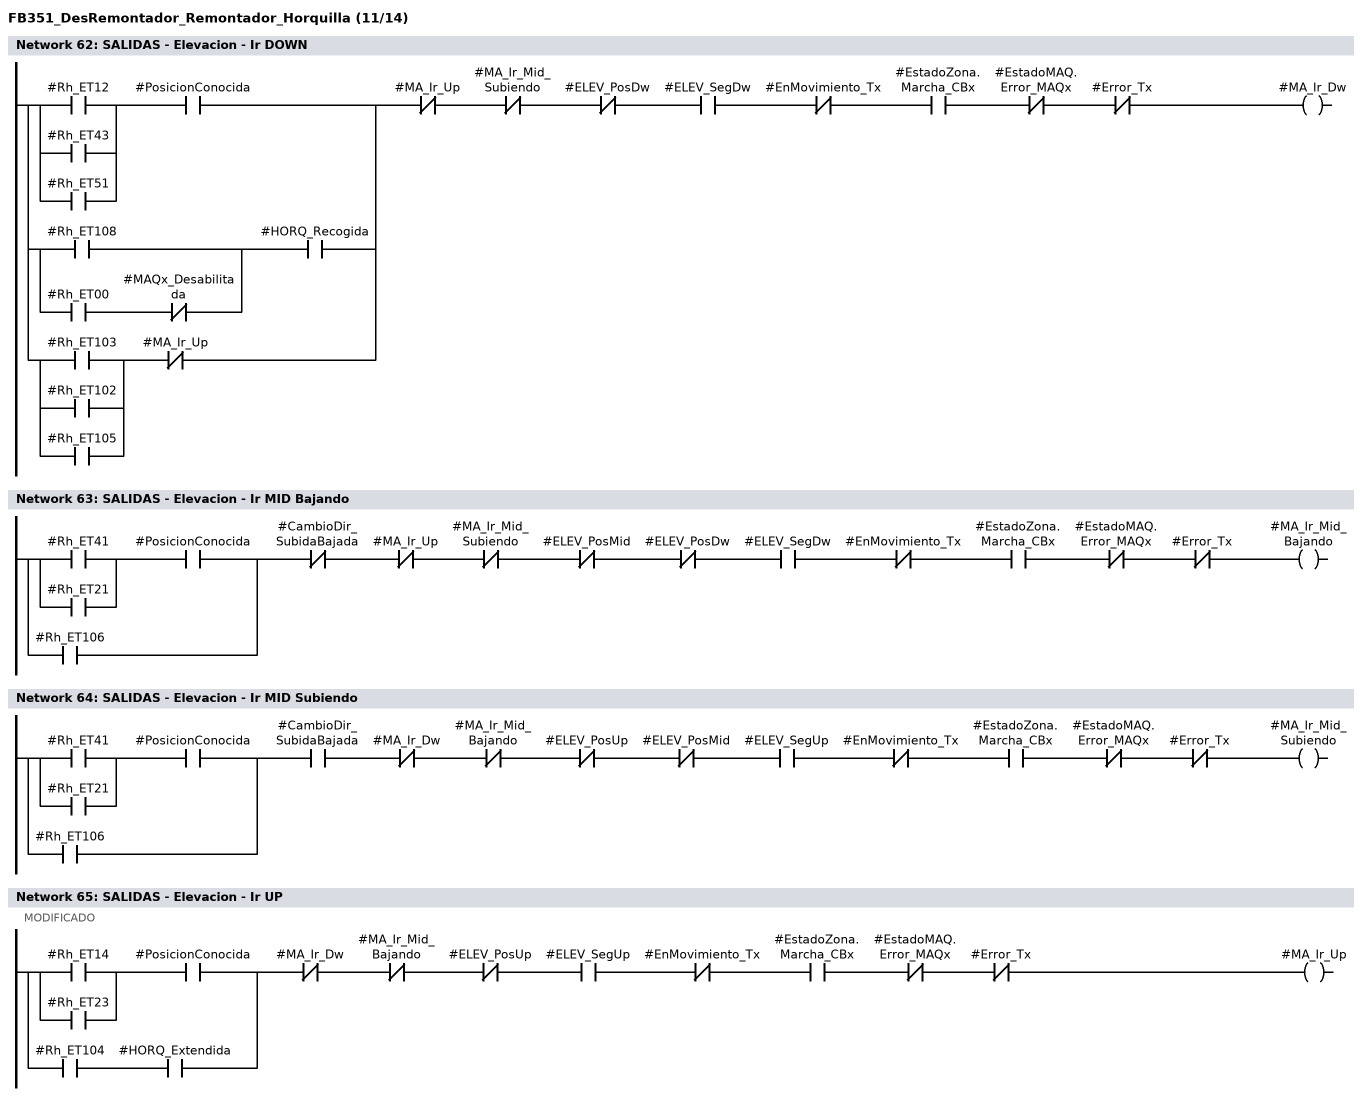
   RUNG wire#powerrail
      Contact( #Rh_ET12 )
      wire#w1
      Contact( #PosicionConocida )
      wire#w2
      I_Contact( #MA_Ir_Up )
      I_Contact( #MA_Ir_Mid_Subiendo )
      I_Contact( #ELEV_PosDw )
      Contact( #ELEV_SegDw )
      I_Contact( #EnMovimiento_Tx )
      Contact( #EstadoZona.Marcha_CBx )
      I_Contact( #EstadoMAQ.Error_MAQx )
      I_Contact( #Error_Tx )
      Coil( #MA_Ir_Dw )
   END_RUNG
   RUNG wire#powerrail
      Contact( #Rh_ET43 )
   END_RUNG wire#w1
   RUNG wire#powerrail
      Contact( #Rh_ET51 )
   END_RUNG wire#w1
   RUNG wire#powerrail
      Contact( #Rh_ET108 )
      wire#w3
      Contact( #HORQ_Recogida )
   END_RUNG wire#w2
   RUNG wire#powerrail
      Contact( #Rh_ET00 )
      I_Contact( #MAQx_Desabilitada )
   END_RUNG wire#w3
   RUNG wire#powerrail
      Contact( #Rh_ET103 )
      wire#w4
      I_Contact( #MA_Ir_Up )
   END_RUNG wire#w2
   RUNG wire#powerrail
      Contact( #Rh_ET102 )
   END_RUNG wire#w4
   RUNG wire#powerrail
      Contact( #Rh_ET105 )
   END_RUNG wire#w4
   // the same network as SCL:
   #MA_Ir_Dw := (((#Rh_ET12 OR #Rh_ET43 OR #Rh_ET51) AND #PosicionConocida) OR ((#Rh_ET108 OR (#Rh_ET00 AND NOT #MAQx_Desabilitada)) AND #HORQ_Recogida) OR ((#Rh_ET103 OR #Rh_ET102 OR #Rh_ET105) AND NOT #MA_Ir_Up)) AND NOT #MA_Ir_Up AND NOT #MA_Ir_Mid_Subiendo AND NOT #ELEV_PosDw AND #ELEV_SegDw AND NOT #EnMovimiento_Tx AND #EstadoZona.Marcha_CBx AND NOT #EstadoMAQ.Error_MAQx AND NOT #Error_Tx;
END_REGION

REGION Network 63: SALIDAS - Elevacion - Ir MID Bajando
   RUNG wire#powerrail
      Contact( #Rh_ET41 )
      wire#w1
      Contact( #PosicionConocida )
      wire#w2
      I_Contact( #CambioDir_SubidaBajada )
      I_Contact( #MA_Ir_Up )
      I_Contact( #MA_Ir_Mid_Subiendo )
      I_Contact( #ELEV_PosMid )
      I_Contact( #ELEV_PosDw )
      Contact( #ELEV_SegDw )
      I_Contact( #EnMovimiento_Tx )
      Contact( #EstadoZona.Marcha_CBx )
      I_Contact( #EstadoMAQ.Error_MAQx )
      I_Contact( #Error_Tx )
      Coil( #MA_Ir_Mid_Bajando )
   END_RUNG
   RUNG wire#powerrail
      Contact( #Rh_ET21 )
   END_RUNG wire#w1
   RUNG wire#powerrail
      Contact( #Rh_ET106 )
   END_RUNG wire#w2
   // the same network as SCL:
   #MA_Ir_Mid_Bajando := (((#Rh_ET41 OR #Rh_ET21) AND #PosicionConocida) OR #Rh_ET106) AND NOT #CambioDir_SubidaBajada AND NOT #MA_Ir_Up AND NOT #MA_Ir_Mid_Subiendo AND NOT #ELEV_PosMid AND NOT #ELEV_PosDw AND #ELEV_SegDw AND NOT #EnMovimiento_Tx AND #EstadoZona.Marcha_CBx AND NOT #EstadoMAQ.Error_MAQx AND NOT #Error_Tx;
END_REGION

REGION Network 64: SALIDAS - Elevacion - Ir MID Subiendo
   RUNG wire#powerrail
      Contact( #Rh_ET41 )
      wire#w1
      Contact( #PosicionConocida )
      wire#w2
      Contact( #CambioDir_SubidaBajada )
      I_Contact( #MA_Ir_Dw )
      I_Contact( #MA_Ir_Mid_Bajando )
      I_Contact( #ELEV_PosUp )
      I_Contact( #ELEV_PosMid )
      Contact( #ELEV_SegUp )
      I_Contact( #EnMovimiento_Tx )
      Contact( #EstadoZona.Marcha_CBx )
      I_Contact( #EstadoMAQ.Error_MAQx )
      I_Contact( #Error_Tx )
      Coil( #MA_Ir_Mid_Subiendo )
   END_RUNG
   RUNG wire#powerrail
      Contact( #Rh_ET21 )
   END_RUNG wire#w1
   RUNG wire#powerrail
      Contact( #Rh_ET106 )
   END_RUNG wire#w2
   // the same network as SCL:
   #MA_Ir_Mid_Subiendo := (((#Rh_ET41 OR #Rh_ET21) AND #PosicionConocida) OR #Rh_ET106) AND #CambioDir_SubidaBajada AND NOT #MA_Ir_Dw AND NOT #MA_Ir_Mid_Bajando AND NOT #ELEV_PosUp AND NOT #ELEV_PosMid AND #ELEV_SegUp AND NOT #EnMovimiento_Tx AND #EstadoZona.Marcha_CBx AND NOT #EstadoMAQ.Error_MAQx AND NOT #Error_Tx;
END_REGION

REGION Network 65: SALIDAS - Elevacion - Ir UP
   // MODIFICADO
   RUNG wire#powerrail
      Contact( #Rh_ET14 )
      wire#w1
      Contact( #PosicionConocida )
      wire#w2
      I_Contact( #MA_Ir_Dw )
      I_Contact( #MA_Ir_Mid_Bajando )
      I_Contact( #ELEV_PosUp )
      Contact( #ELEV_SegUp )
      I_Contact( #EnMovimiento_Tx )
      Contact( #EstadoZona.Marcha_CBx )
      I_Contact( #EstadoMAQ.Error_MAQx )
      I_Contact( #Error_Tx )
      Coil( #MA_Ir_Up )
   END_RUNG
   RUNG wire#powerrail
      Contact( #Rh_ET23 )
   END_RUNG wire#w1
   RUNG wire#powerrail
      Contact( #Rh_ET104 )
      Contact( #HORQ_Extendida )
   END_RUNG wire#w2
   // the same network as SCL:
   #MA_Ir_Up := (((#Rh_ET14 OR #Rh_ET23) AND #PosicionConocida) OR (#Rh_ET104 AND #HORQ_Extendida)) AND NOT #MA_Ir_Dw AND NOT #MA_Ir_Mid_Bajando AND NOT #ELEV_PosUp AND #ELEV_SegUp AND NOT #EnMovimiento_Tx AND #EstadoZona.Marcha_CBx AND NOT #EstadoMAQ.Error_MAQx AND NOT #Error_Tx;
END_REGION

REGION Network 66: SALIDAS - Hoquilla - Velocidad Rapida
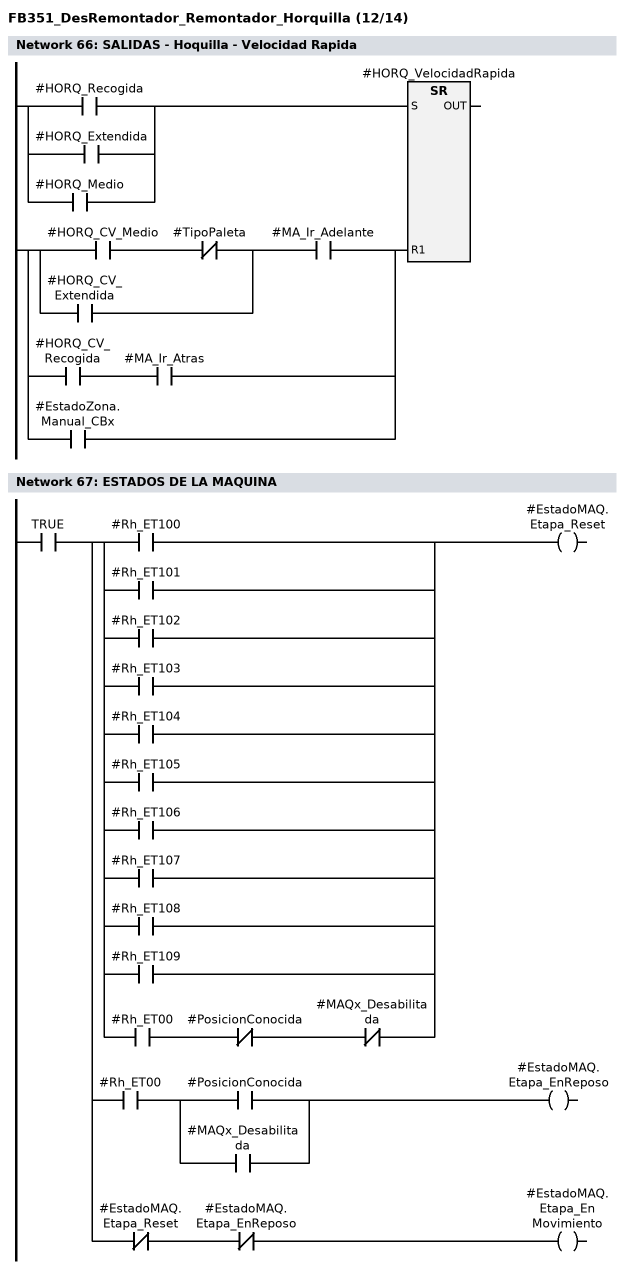
   RUNG wire#powerrail
      Contact( #HORQ_Recogida )
      wire#w1
      S_SR(operand := #HORQ_VelocidadRapida, r1 := wire#w3)
   END_RUNG
   RUNG wire#powerrail
      Contact( #HORQ_Extendida )
   END_RUNG wire#w1
   RUNG wire#powerrail
      Contact( #HORQ_Medio )
   END_RUNG wire#w1
   RUNG wire#powerrail
      Contact( #HORQ_CV_Medio )
      I_Contact( #TipoPaleta )
      wire#w2
      Contact( #MA_Ir_Adelante )
   END_RUNG wire#w3
   RUNG wire#powerrail
      Contact( #HORQ_CV_Extendida )
   END_RUNG wire#w2
   RUNG wire#powerrail
      Contact( #HORQ_CV_Recogida )
      Contact( #MA_Ir_Atras )
   END_RUNG wire#w3
   RUNG wire#powerrail
      Contact( #EstadoZona.Manual_CBx )
   END_RUNG wire#w3
   // the same network as SCL:
   IF #HORQ_Recogida OR #HORQ_Extendida OR #HORQ_Medio THEN
       #HORQ_VelocidadRapida := TRUE;   // SR flip-flop
   END_IF;
   IF (((#HORQ_CV_Medio AND NOT #TipoPaleta) OR #HORQ_CV_Extendida) AND #MA_Ir_Adelante) OR (#HORQ_CV_Recogida AND #MA_Ir_Atras) OR #EstadoZona.Manual_CBx THEN
       #HORQ_VelocidadRapida := FALSE;
   END_IF;
END_REGION

REGION Network 67: ESTADOS DE LA MAQUINA
   RUNG wire#powerrail
      Contact( TRUE )
      wire#w1
      Contact( #Rh_ET100 )
      wire#w2
      Coil( #EstadoMAQ.Etapa_Reset )
   END_RUNG
   RUNG wire#w1
      Contact( #Rh_ET101 )
   END_RUNG wire#w2
   RUNG wire#w1
      Contact( #Rh_ET102 )
   END_RUNG wire#w2
   RUNG wire#w1
      Contact( #Rh_ET103 )
   END_RUNG wire#w2
   RUNG wire#w1
      Contact( #Rh_ET104 )
   END_RUNG wire#w2
   RUNG wire#w1
      Contact( #Rh_ET105 )
   END_RUNG wire#w2
   RUNG wire#w1
      Contact( #Rh_ET106 )
   END_RUNG wire#w2
   RUNG wire#w1
      Contact( #Rh_ET107 )
   END_RUNG wire#w2
   RUNG wire#w1
      Contact( #Rh_ET108 )
   END_RUNG wire#w2
   RUNG wire#w1
      Contact( #Rh_ET109 )
   END_RUNG wire#w2
   RUNG wire#w1
      Contact( #Rh_ET00 )
      I_Contact( #PosicionConocida )
      I_Contact( #MAQx_Desabilitada )
   END_RUNG wire#w2
   RUNG wire#w1
      Contact( #Rh_ET00 )
      wire#w3
      Contact( #PosicionConocida )
      wire#w4
      Coil( #EstadoMAQ.Etapa_EnReposo )
   END_RUNG
   RUNG wire#w3
      Contact( #MAQx_Desabilitada )
   END_RUNG wire#w4
   RUNG wire#w1
      I_Contact( #EstadoMAQ.Etapa_Reset )
      I_Contact( #EstadoMAQ.Etapa_EnReposo )
      Coil( #EstadoMAQ.Etapa_EnMovimiento )
   END_RUNG
   // the same network as SCL:
   #EstadoMAQ.Etapa_Reset := TRUE AND (#Rh_ET100 OR #Rh_ET101 OR #Rh_ET102 OR #Rh_ET103 OR #Rh_ET104 OR #Rh_ET105 OR #Rh_ET106 OR #Rh_ET107 OR #Rh_ET108 OR #Rh_ET109 OR (#Rh_ET00 AND NOT #PosicionConocida AND NOT #MAQx_Desabilitada));
   #EstadoMAQ.Etapa_EnReposo := TRUE AND #Rh_ET00 AND (#PosicionConocida OR #MAQx_Desabilitada);
   #EstadoMAQ.Etapa_EnMovimiento := TRUE AND NOT #EstadoMAQ.Etapa_Reset AND NOT #EstadoMAQ.Etapa_EnReposo;
END_REGION

REGION Network 68: ENTRADAS DE LA MAQUINA
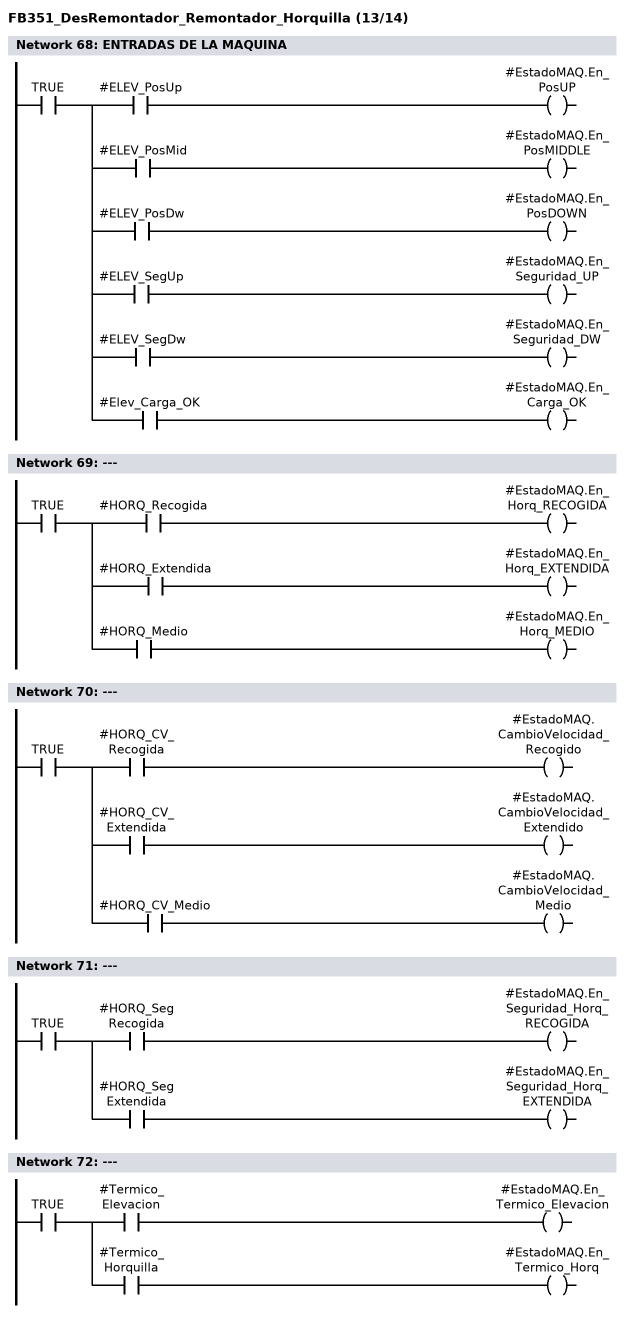
   RUNG wire#powerrail
      Contact( TRUE )
      wire#w1
      Contact( #ELEV_PosUp )
      Coil( #EstadoMAQ.En_PosUP )
   END_RUNG
   RUNG wire#w1
      Contact( #ELEV_PosMid )
      Coil( #EstadoMAQ.En_PosMIDDLE )
   END_RUNG
   RUNG wire#w1
      Contact( #ELEV_PosDw )
      Coil( #EstadoMAQ.En_PosDOWN )
   END_RUNG
   RUNG wire#w1
      Contact( #ELEV_SegUp )
      Coil( #EstadoMAQ.En_Seguridad_UP )
   END_RUNG
   RUNG wire#w1
      Contact( #ELEV_SegDw )
      Coil( #EstadoMAQ.En_Seguridad_DW )
   END_RUNG
   RUNG wire#w1
      Contact( #Elev_Carga_OK )
      Coil( #EstadoMAQ.En_Carga_OK )
   END_RUNG
   // the same network as SCL:
   #EstadoMAQ.En_PosUP := TRUE AND #ELEV_PosUp;
   #EstadoMAQ.En_PosMIDDLE := TRUE AND #ELEV_PosMid;
   #EstadoMAQ.En_PosDOWN := TRUE AND #ELEV_PosDw;
   #EstadoMAQ.En_Seguridad_UP := TRUE AND #ELEV_SegUp;
   #EstadoMAQ.En_Seguridad_DW := TRUE AND #ELEV_SegDw;
   #EstadoMAQ.En_Carga_OK := TRUE AND #Elev_Carga_OK;
END_REGION

REGION Network 69: ---
   RUNG wire#powerrail
      Contact( TRUE )
      wire#w1
      Contact( #HORQ_Recogida )
      Coil( #EstadoMAQ.En_Horq_RECOGIDA )
   END_RUNG
   RUNG wire#w1
      Contact( #HORQ_Extendida )
      Coil( #EstadoMAQ.En_Horq_EXTENDIDA )
   END_RUNG
   RUNG wire#w1
      Contact( #HORQ_Medio )
      Coil( #EstadoMAQ.En_Horq_MEDIO )
   END_RUNG
   // the same network as SCL:
   #EstadoMAQ.En_Horq_RECOGIDA := TRUE AND #HORQ_Recogida;
   #EstadoMAQ.En_Horq_EXTENDIDA := TRUE AND #HORQ_Extendida;
   #EstadoMAQ.En_Horq_MEDIO := TRUE AND #HORQ_Medio;
END_REGION

REGION Network 70: ---
   RUNG wire#powerrail
      Contact( TRUE )
      wire#w1
      Contact( #HORQ_CV_Recogida )
      Coil( #EstadoMAQ.CambioVelocidad_Recogido )
   END_RUNG
   RUNG wire#w1
      Contact( #HORQ_CV_Extendida )
      Coil( #EstadoMAQ.CambioVelocidad_Extendido )
   END_RUNG
   RUNG wire#w1
      Contact( #HORQ_CV_Medio )
      Coil( #EstadoMAQ.CambioVelocidad_Medio )
   END_RUNG
   // the same network as SCL:
   #EstadoMAQ.CambioVelocidad_Recogido := TRUE AND #HORQ_CV_Recogida;
   #EstadoMAQ.CambioVelocidad_Extendido := TRUE AND #HORQ_CV_Extendida;
   #EstadoMAQ.CambioVelocidad_Medio := TRUE AND #HORQ_CV_Medio;
END_REGION

REGION Network 71: ---
   RUNG wire#powerrail
      Contact( TRUE )
      wire#w1
      Contact( #HORQ_SegRecogida )
      Coil( #EstadoMAQ.En_Seguridad_Horq_RECOGIDA )
   END_RUNG
   RUNG wire#w1
      Contact( #HORQ_SegExtendida )
      Coil( #EstadoMAQ.En_Seguridad_Horq_EXTENDIDA )
   END_RUNG
   // the same network as SCL:
   #EstadoMAQ.En_Seguridad_Horq_RECOGIDA := TRUE AND #HORQ_SegRecogida;
   #EstadoMAQ.En_Seguridad_Horq_EXTENDIDA := TRUE AND #HORQ_SegExtendida;
END_REGION

REGION Network 72: ---
   RUNG wire#powerrail
      Contact( TRUE )
      wire#w1
      Contact( #Termico_Elevacion )
      Coil( #EstadoMAQ.En_Termico_Elevacion )
   END_RUNG
   RUNG wire#w1
      Contact( #Termico_Horquilla )
      Coil( #EstadoMAQ.En_Termico_Horq )
   END_RUNG
   // the same network as SCL:
   #EstadoMAQ.En_Termico_Elevacion := TRUE AND #Termico_Elevacion;
   #EstadoMAQ.En_Termico_Horq := TRUE AND #Termico_Horquilla;
END_REGION

REGION Network 73: SALIDAS DE LA MAQUINA
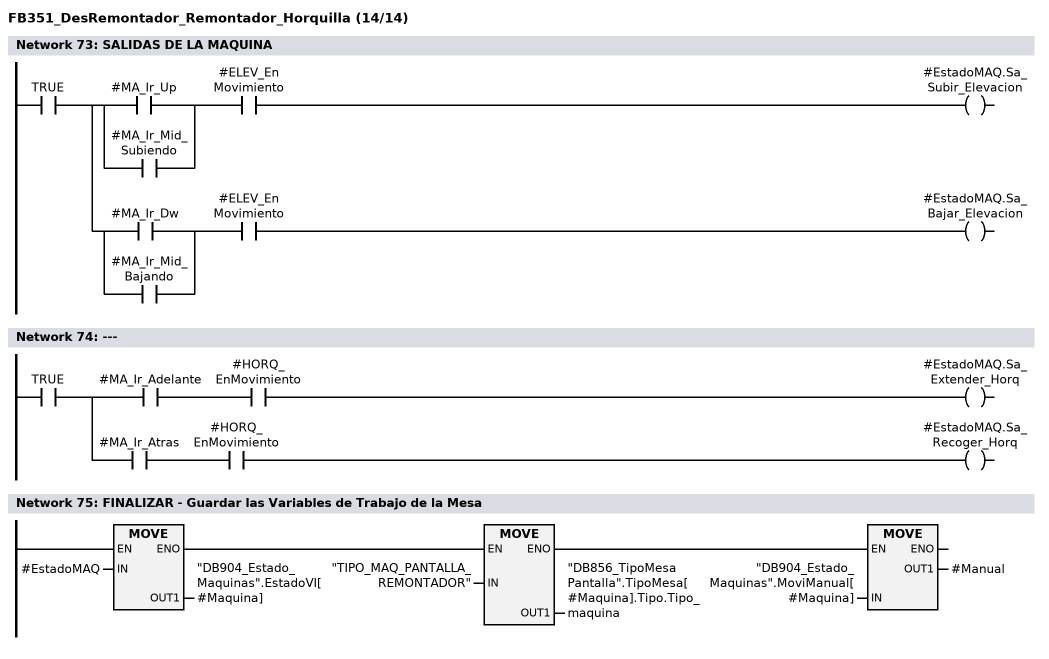
   RUNG wire#powerrail
      Contact( TRUE )
      wire#w1
      Contact( #MA_Ir_Up )
      wire#w2
      Contact( #ELEV_EnMovimiento )
      Coil( #EstadoMAQ.Sa_Subir_Elevacion )
   END_RUNG
   RUNG wire#w1
      Contact( #MA_Ir_Mid_Subiendo )
   END_RUNG wire#w2
   RUNG wire#w1
      Contact( #MA_Ir_Dw )
      wire#w3
      Contact( #ELEV_EnMovimiento )
      Coil( #EstadoMAQ.Sa_Bajar_Elevacion )
   END_RUNG
   RUNG wire#w1
      Contact( #MA_Ir_Mid_Bajando )
   END_RUNG wire#w3
   // the same network as SCL:
   #EstadoMAQ.Sa_Subir_Elevacion := TRUE AND (#MA_Ir_Up OR #MA_Ir_Mid_Subiendo) AND #ELEV_EnMovimiento;
   #EstadoMAQ.Sa_Bajar_Elevacion := TRUE AND (#MA_Ir_Dw OR #MA_Ir_Mid_Bajando) AND #ELEV_EnMovimiento;
END_REGION

REGION Network 74: ---
   RUNG wire#powerrail
      Contact( TRUE )
      wire#w1
      Contact( #MA_Ir_Adelante )
      Contact( #HORQ_EnMovimiento )
      Coil( #EstadoMAQ.Sa_Extender_Horq )
   END_RUNG
   RUNG wire#w1
      Contact( #MA_Ir_Atras )
      Contact( #HORQ_EnMovimiento )
      Coil( #EstadoMAQ.Sa_Recoger_Horq )
   END_RUNG
   // the same network as SCL:
   #EstadoMAQ.Sa_Extender_Horq := TRUE AND #MA_Ir_Adelante AND #HORQ_EnMovimiento;
   #EstadoMAQ.Sa_Recoger_Horq := TRUE AND #MA_Ir_Atras AND #HORQ_EnMovimiento;
END_REGION

REGION Network 75: FINALIZAR - Guardar las Variables de Trabajo de la Mesa
   RUNG wire#powerrail
      Move(in := #EstadoMAQ, out1 => "DB904_Estado_Maquinas".EstadoVI[#Maquina])
      Move(in := "TIPO_MAQ_PANTALLA_REMONTADOR", out1 => "DB856_TipoMesaPantalla".TipoMesa[#Maquina].Tipo.Tipo_maquina)
      Move(in := "DB904_Estado_Maquinas".MoviManual[#Maquina], out1 => #Manual)
   END_RUNG
   // the same network as SCL:
   "DB904_Estado_Maquinas".EstadoVI[#Maquina] := #EstadoMAQ;
   "DB856_TipoMesaPantalla".TipoMesa[#Maquina].Tipo.Tipo_maquina := "TIPO_MAQ_PANTALLA_REMONTADOR";
   #Manual := "DB904_Estado_Maquinas".MoviManual[#Maquina];
END_REGION
END_FUNCTION_BLOCK
